# B&R Automation Studio project NAELD004C00R10L518F00 (part 28)

#### Local.var
```iecst
(*2019-06-07*)
(**)
(*Local Action, State & Status*)
VAR
	eAct : eBufferAction := BufferActIdle;
	eStat : eBufferAction := BufferActIdle;
	eStatus : eFBStatus := Idle;
	udiStatus : UDINT := 0;
	sStatTxt : STRING[200] := '';
	a_sStatText : ARRAY[0..50] OF STRING[200] := ['Idling','Creating Directory','Getting Retained Buffer Data','Setting Buffer Full','Setting Buffer Empty','Loading Board','Loading Board With Slot Check','Unloading Board','Unloading Board With Slot Check','Unloading Board With Cooling Time Check','Unloading Board With Slot Check And Cooling Time Check','Getting Next Load Board Slot Number','Getting Next Load Good Board Slot Number','Getting Next Load Bad Board Slot Number','Getting Next Unload Board Slot Number','Getting Next Unload Good Board Slot Number','Getting Next Unload Bad Board Slot Number','Checking Cooling Time','Checking Cooling Board','Checking Cooling Good Board','Checking Cooling Bad Board','Resetting Buffer','Turning On Cooling Fan','Turning Off Cooling Fan','Background Starting Buffer Set Full','Background Starting Buffer Set Empty','Background Stopping Buffer Set','Background Starting Update Sensor','Background Stopping Update Sensor','Background Starting Update Display','Background Stopping Update Display','Background Starting Cooling Fan','Background Stopping Cooling Fan',18('')];
END_VAR
(**)
(*Local Alarm*)
VAR
	tyAlmData : tyAlmDat;
	a_tyAlmText : ARRAY[10000..10099] OF tyAlmTxt := [(sAlmText:='Create User Directory Error',sRcyText:='An Error Occurred While Attempting To Create User Directory. Please Contact Nutek For A Possible Solution'),(sAlmText:='Create Retain Directory Error',sRcyText:='An Error Occurred While Attempting To Create Retain Directory. Please Contact Nutek For A Possible Solution'),(sAlmText:='File Open Error While Reading Retain File',sRcyText:='An Error Was Encountered While Trying To Open File. Please Contact Nutek For A Possible Solution.'),(sAlmText:='File Read Error While Reading Retain File',sRcyText:='An Error Was Encountered While Trying To Read File. Please Contact Nutek For A Possible Solution.'),(sAlmText:='File Close Error While Reading Retain File',sRcyText:='An Error Was Encountered While Trying To Close File. Please Contact Nutek For A Possible Solution.'),(sAlmText:='File Open Error While Setting Full Buffer',sRcyText:='An Error Was Encountered While Trying To Open File. Please Contact Nutek For A Possible Solution.'),(sAlmText:='File Create Error While Setting Full Buffer',sRcyText:='An Error Was Encountered While Trying To Create File. Please Contact Nutek For A Possible Solution.'),(sAlmText:='File Write Error While Setting Full Buffer',sRcyText:='An Error Was Encountered While Trying To Write File. Please Contact Nutek For A Possible Solution.'),(sAlmText:='File Close Error While Setting Full Buffer',sRcyText:='An Error Was Encountered While Trying To Close File. Please Contact Nutek For A Possible Solution.'),(sAlmText:='File Open Error While Setting Empty Buffer',sRcyText:='An Error Was Encountered While Trying To Open File. Please Contact Nutek For A Possible Solution.'),(sAlmText:='File Create Error While Setting Empty Buffer',sRcyText:='An Error Was Encountered While Trying To Create File. Please Contact Nutek For A Possible Solution.'),(sAlmText:='File Write Error While Setting Empty Buffer',sRcyText:='An Error Was Encountered While Trying To Write File. Please Contact Nutek For A Possible Solution.'),(sAlmText:='File Close Error While Setting Empty Buffer',sRcyText:='An Error Was Encountered While Trying To Close File. Please Contact Nutek For A Possible Solution.'),(sAlmText:='File Open Error While Loading Info To Buffer',sRcyText:='An Error Was Encountered While Trying To Open File. Please Contact Nutek For A Possible Solution.'),(sAlmText:='File Create Error While Loading Info To Buffer',sRcyText:='An Error Was Encountered While Trying To Create File. Please Contact Nutek For A Possible Solution.'),(sAlmText:='File Write Error While Loading Info To Buffer',sRcyText:='An Error Was Encountered While Trying To Write File. Please Contact Nutek For A Possible Solution.'),(sAlmText:='File Close Error While Loading Info To Buffer',sRcyText:='An Error Was Encountered While Trying To Close File. Please Contact Nutek For A Possible Solution.'),(sAlmText:='Wrong Slot Number To Load',sRcyText:='Invalid Slot to Load The Board.'),(sAlmText:='File Open Error While Loading Info To Buffer With Slot Check',sRcyText:='An Error Was Encountered While Trying To Open File. Please Contact Nutek For A Possible Solution.'),(sAlmText:='File Create Error While Loading Info To Buffer With Slot Check',sRcyText:='An Error Was Encountered While Trying To Create File. Please Contact Nutek For A Possible Solution.'),(sAlmText:='File Write Error While Loading Info To Buffer With Slot Check',sRcyText:='An Error Was Encountered While Trying To Write File. Please Contact Nutek For A Possible Solution.'),(sAlmText:='File Close Error While Loading Info To Buffer With Slot Check',sRcyText:='An Error Was Encountered While Trying To Close File. Please Contact Nutek For A Possible Solution.'),(sAlmText:='File Open Error While Unloading Info From Buffer',sRcyText:='An Error Was Encountered While Trying To Open File. Please Contact Nutek For A Possible Solution.'),(sAlmText:='File Create Error While Unloading Info From Buffer',sRcyText:='An Error Was Encountered While Trying To Create File. Please Contact Nutek For A Possible Solution.'),(sAlmText:='File Write Error While Unloading Info From Buffer',sRcyText:='An Error Was Encountered While Trying To Write File. Please Contact Nutek For A Possible Solution.'),(sAlmText:='File Close Error While Unloading Info From Buffer',sRcyText:='An Error Was Encountered While Trying To Close File. Please Contact Nutek For A Possible Solution.'),(sAlmText:='Wrong Slot Number To Unload',sRcyText:='Invalid Slot to Unload The Board.'),(sAlmText:='File Open Error While Unloading Info From Buffer With Slot Check',sRcyText:='An Error Was Encountered While Trying To Open File. Please Contact Nutek For A Possible Solution.'),(sAlmText:='File Create Error While Unloading Info From Buffer With Slot Check',sRcyText:='An Error Was Encountered While Trying To Create File. Please Contact Nutek For A Possible Solution.'),(sAlmText:='File Write Error While Unloading Info From Buffer With Slot Check',sRcyText:='An Error Was Encountered While Trying To Write File. Please Contact Nutek For A Possible Solution.'),(sAlmText:='File Close Error While Unloading Info From Buffer With Slot Check',sRcyText:='An Error Was Encountered While Trying To Close File. Please Contact Nutek For A Possible Solution.'),(sAlmText:='File Open Error While Unloading Info From Buffer With Cooling Time Check',sRcyText:='An Error Was Encountered While Trying To Open File. Please Contact Nutek For A Possible Solution.'),(sAlmText:='File Create Error While Unloading Info From Buffer With Cooling Time Check',sRcyText:='An Error Was Encountered While Trying To Create File. Please Contact Nutek For A Possible Solution.'),(sAlmText:='File Write Error While Unloading Info From Buffer With Cooling Time Check',sRcyText:='An Error Was Encountered While Trying To Write File. Please Contact Nutek For A Possible Solution.'),(sAlmText:='File Close Error While Unloading Info From Buffer With Cooling Time Check',sRcyText:='An Error Was Encountered While Trying To Close File. Please Contact Nutek For A Possible Solution.'),(sAlmText:='Wrong Slot Number To Unload With Cooling Time Check',sRcyText:='Invalid Slot to Unload The Board with Cooling Time Check.'),(sAlmText:='File Open Error While Unloading Info From Buffer With Slot Check And Cooling Time Check',sRcyText:='An Error Was Encountered While Trying To Open File. Please Contact Nutek For A Possible Solution.'),(sAlmText:='File Create Error While Unloading Info From Buffer With Slot Check And Cooling Time Check',sRcyText:='An Error Was Encountered While Trying To Create File. Please Contact Nutek For A Possible Solution.'),(sAlmText:='File Write Error While Unloading Info From Buffer With Slot Check And Cooling Time Check',sRcyText:='An Error Was Encountered While Trying To Write File. Please Contact Nutek For A Possible Solution.'),(sAlmText:='File Close Error While Unloading Info From Buffer With Slot Check And Cooling Time Check',sRcyText:='An Error Was Encountered While Trying To Close File. Please Contact Nutek For A Possible Solution.'),(sAlmText:='Directory Does Not Exist While Setting Full Buffer',sRcyText:='The Directory Does Not Exist. Please Contact Nutek For A Possible Solution.'),(sAlmText:='Directory Does Not Exist While Setting Empty Buffer',sRcyText:='The Directory Does Not Exist. Please Contact Nutek For A Possible Solution.'),(sAlmText:='Directory Does Not Exist While Loading Info To Buffer',sRcyText:='The Directory Does Not Exist. Please Contact Nutek For A Possible Solution.'),(sAlmText:='Directory Does Not Exist While Loading Info To Buffer With Slot Check',sRcyText:='The Directory Does Not Exist. Please Contact Nutek For A Possible Solution.'),(sAlmText:='Directory Does Not Exist While Unloading Info From Buffer',sRcyText:='The Directory Does Not Exist. Please Contact Nutek For A Possible Solution.'),(sAlmText:='Directory Does Not Exist While Unloading Info From Buffer With Slot Check',sRcyText:='The Directory Does Not Exist. Please Contact Nutek For A Possible Solution.'),(sAlmText:='Directory Does Not Exist While Unloading Info From Buffer With Cooling Time Check',sRcyText:='The Directory Does Not Exist. Please Contact Nutek For A Possible Solution.'),(sAlmText:='Directory Does Not Exist While Unloading Info From Buffer With Slot Check And Cooling Time Check',sRcyText:='The Directory Does Not Exist. Please Contact Nutek For A Possible Solution.'),(sAlmText:='Unloading Slot Is Skipped While Unloading Buffer',sRcyText:='Unload From Wrong Slot (Skip Slot).'),(sAlmText:='Unloading Slot Is Not For Board While Unloading Buffer',sRcyText:='Unload From Wrong Slot (Not For Board).'),(sAlmText:='Unloading Slot Board Is Not Available While Unloading Buffer',sRcyText:='Unload From Wrong Slot (Board Is Not Available).'),(sAlmText:='Unloading Last Sub Slot Is Not For Board While Unloading Buffer',sRcyText:='Unload From Wrong Slot (Last Sub Slot Is Not For Board).'),(sAlmText:='Unloading Last Sub Slot Has No Board While Unloading Buffer',sRcyText:='Unload From Wrong Slot (Last Sub Slot Has No Board).'),(sAlmText:='Board Quantity In Slot Is 0 While Unloading Buffer',sRcyText:='Unload From Wrong Slot (Board Quantity In Slot = 0).'),(sAlmText:='Board Capacity In Slot Is 0 While Unloading Buffer',sRcyText:='Unload From Wrong Slot (Board Capacity In Slot = 0).'),(sAlmText:='Unloading Slot Is Skipped While Unloading Buffer With Slot Check',sRcyText:='Unload From Wrong Slot (Skip Slot).'),(sAlmText:='Unloading Slot Is Not For Board While Unloading Buffer With Slot Check',sRcyText:='Unload From Wrong Slot (Not For Board).'),(sAlmText:='Unloading Slot Board Is Not available While Unloading Buffer With Slot Check',sRcyText:='Unload From Wrong Slot (Board Is Not Available).'),(sAlmText:='Unloading Last Sub Slot Is Not For Board While Unloading Buffer With Slot Check',sRcyText:='Unload From Wrong Slot (Last Sub Slot Is Not For Board).'),(sAlmText:='Unloading Last Sub Slot Has No Board While Unloading Buffer With Slot Check',sRcyText:='Unload From Wrong Slot (Last Sub Slot Has No Board).'),(sAlmText:='Board Quantity In Slot Is 0 While Unloading Buffer With Slot Check',sRcyText:='Unload From Wrong Slot (Board Quantity In Slot = 0).'),(sAlmText:='Board Capacity In Slot Is 0 While Unloading Buffer With Slot Check',sRcyText:='Unload From Wrong Slot (Board Capacity In Slot = 0).'),(sAlmText:='Unloading Slot Is Skipped While Unloading Buffer With Cool Check',sRcyText:='Unload From Wrong Slot (Skip Slot).'),(sAlmText:='Unloading Slot Is Not For Board While Unloading Buffer With Cool Check',sRcyText:='Unload From Wrong Slot (Not For Board).'),(sAlmText:='Unloading Slot Board Is Not available While Unloading Buffer With Cool Check',sRcyText:='Unload From Wrong Slot (Board Is Not Available).'),(sAlmText:='Unloading Last Sub Slot Is Not For Board While Unloading Buffer With Cool Check',sRcyText:='Unload From Wrong Slot (Last Sub Slot Is Not For Board).'),(sAlmText:='Unloading Last Sub Slot Has No Board While Unloading Buffer With Cool Check',sRcyText:='Unload From Wrong Slot (Last Sub Slot Has No Board).'),(sAlmText:='Board Quantity In Slot Is 0 While Unloading Buffer With Cool Check',sRcyText:='Unload From Wrong Slot (Board Quantity In Slot = 0).'),(sAlmText:='Board Capacity In Slot Is 0 While Unloading Buffer With Cool Check',sRcyText:='Unload From Wrong Slot (Board Capacity In Slot = 0).'),(sAlmText:='Unloading Slot Is Skipped While Unloading Buffer With Cool & Slot Check',sRcyText:='Unload From Wrong Slot (Skip Slot).'),(sAlmText:='Unloading Slot Is Not For Board While Unloading Buffer With Cool & Slot Check',sRcyText:='Unload From Wrong Slot (Not For Board).'),(sAlmText:='Unloading Slot Board Is Not available While Unloading Buffer With Cool & Slot Check',sRcyText:='Unload From Wrong Slot (Board Is Not Available).'),(sAlmText:='Unloading Last Sub Slot Is Not For Board While Unloading Buffer With Cool & Slot Check',sRcyText:='Unload From Wrong Slot (Last Sub Slot Is Not For Board).'),(sAlmText:='Unloading Last Sub Slot Has No Board While Unloading Buffer With Cool & Slot Check',sRcyText:='Unload From Wrong Slot (Last Sub Slot Has No Board).'),(sAlmText:='Board Quantity In Slot Is 0 While Unloading Buffer With Cool & Slot Check',sRcyText:='Unload From Wrong Slot (Board Quantity In Slot = 0).'),(sAlmText:='Board Capacity In Slot Is 0 While Unloading Buffer With Cool & Slot Check',sRcyText:='Unload From Wrong Slot (Board Capacity In Slot = 0).'),(sAlmText:='Loading Slot Is Not For Board',sRcyText:='Load To Wrong Slot (Not For Board).'),(sAlmText:='Loading Slot Is Full Of Board',sRcyText:='Load To Wrong Slot (Full With Board).'),(sAlmText:='Loading First Sub-Slot Is Not For Board',sRcyText:='Load To Wrong Slot (First Sub Slot Not For Board).'),(sAlmText:='Loading Last Sub-Slot Have Board, Which Mean Slot Is Full Of Board',sRcyText:='Load To Wrong Slot (Full With Board(Last Sub Slot Have Board)).'),(sAlmText:='Loading Last Sub-Slot Is Not For Board',sRcyText:='Load To Wrong Slot (Last Sub Slot Not For Board).'),(sAlmText:='Loading Slot Is Full Of Board',sRcyText:='Load To Wrong Slot (Full With Board).'),(sAlmText:='Loading Slot Is Skipped',sRcyText:='Load To Wrong Slot (Skip Slot).'),(sAlmText:='Existing Board Status Is Different With Loading Board Status',sRcyText:='Existing Board Status Is Different With Loading Buffer Status.'),(sAlmText:='Loading Slot Is Not For Board',sRcyText:='Load To Wrong Slot (Not For Board).'),(sAlmText:='Loading Slot Is Full Of Board',sRcyText:='Load To Wrong Slot (Full With Board).'),(sAlmText:='Loading First Sub-Slot Is Not For Board',sRcyText:='Load To Wrong Slot (First Sub Slot Not For Board).'),(sAlmText:='Loading Last Sub-Slot Have Board, Which Mean Slot Is Full Of Board',sRcyText:='Load To Wrong Slot (Full With Board(Last Sub Slot Have Board)).'),(sAlmText:='Loading Last Sub-Slot Is Not For Board',sRcyText:='Load To Wrong Slot (Last Sub Slot Not For Board).'),(sAlmText:='Loading Slot Is Full Of Board',sRcyText:='Load To Wrong Slot (Full With Board).'),(sAlmText:='Loading Slot Is Skipped',sRcyText:='Load To Wrong Slot (Skip Slot).'),(sAlmText:='Existing Board Status Is Different With Loading Board Status',sRcyText:='Existing Board Status Is Different With Loading Buffer Status.'),8((0))];
END_VAR
(**)
(*Local Output*)
VAR
	diNxtLoadSlt : DINT;
	diNxtUnloadSlt : DINT;
	diCoolBrdAny : DINT;
	diCoolBrdGd : DINT;
	diCoolBrdBad : DINT;
	bCoolNotRdy : BOOL;
	tyBuffer : tyBffr;
	tyDispBuffer : tyDispBffr;
	tyBufferStat : tyBffrStat;
	tyBoardUnloadStat : tyBrdUnloadStat;
	bFileNotFound : BOOL;
	bCoolFanCtrl : BOOL;
END_VAR
VAR RETAIN
	bMagPresent : BOOL;
END_VAR
VAR
	dtMagPresentTm : DATE_AND_TIME;
	bNewProduct : BOOL;
	bLastProductUnload : BOOL;
	bLastProductLeftInBffr : BOOL;
	bParamDiff : BOOL;
	bMagRemoved : BOOL;
	bFIFOOld : BOOL;
END_VAR
(**)
(*Local Input*)
VAR
	udiRstErr : UDINT := 0;
	sFileName : STRING[80] := 'Buffer.dat';
	bManual : BOOL := FALSE;
	dtCurrDT : DATE_AND_TIME;
	diMinSlt : DINT;
	diMaxSlt : DINT;
	diPitch : DINT;
	diSltCap : DINT := 1;
	diBffrTtlSlt : DINT;
	diCoolTm : DINT;
	diSltToSltInUM : DINT;
	diLifterBtmPosInUM : DINT;
	diLifterCurrPosInUM : DINT;
	bAscending : BOOL;
	bFIFO : BOOL;
	bGdBrdIn : BOOL;
	bGdBrdReq : BOOL;
	bNxtLoadSeq : BOOL;
	a_bSkip : ARRAY[1..c_diBffrSize] OF BOOL;
	diCoolFanOffDlyTm : DINT := 30000;
	bMagPresentSensor : BOOL;
	bPrepCoolFan : BOOL := TRUE;
	bCoolFanTm : BOOL := TRUE;
	sBffrNm : STRING[15];
	sProdNm : STRING[15];
	sBarcode1 : STRING[80];
	sBarcode2 : STRING[80];
	sCurrRcpNm : {REDUND_UNREPLICABLE} STRING[15];
	sProgNm : STRING[15] := 'Buffer';
	bNtSettingsLoadDone : BOOL := TRUE;
END_VAR
(**)
(*Local*)
VAR
	bRstErr : BOOL;
	udiRstErrOld : UDINT;
	bInitDone : BOOL;
	bInitialDone : BOOL;
	bUpdateSensor : BOOL;
	bBffrSetMty : BOOL;
	bBffrSetFull : BOOL;
	bUpdtDisplay : BOOL;
	usiStep : USINT;
	diCurrSlt : DINT;
	diExpectedSlt : DINT;
	bSetFull : BOOL;
	bSetMty : BOOL;
	bCoolFanRun : BOOL;
	tyBffrParameter : tyBffrParam;
	fbDirCreate1 : fbDirCreate;
	fbDirCreate2 : fbDirCreate;
	fbFileRead1 : fbFileFullRead;
	fbFileWrite1 : fbFileFullWrite;
	fbCoolFanOffDlyTm : TON;
	fbCoolFanOffChkTm : TON := (PT:=T#500ms);
	fbMagAbsentTm : TON := (PT:=T#5s);
	fbMagPresentTm : TON := (PT:=T#8s);
	eStatOld : eBufferAction := BufferActIdle;
	udiModuleNum : UDINT := 2001;
END_VAR
```

#### Act_Alarm.st
```iecst
(** 2019-03-25 **)
ACTION Act_Alarm:

	//Error
	IF EDGEPOS(eStatus = Error) THEN

		tyAlmData.sProgNm		:= p_sProgNm;
		tyAlmData.udiCode		:= udiStatus;
		tyAlmData.eSeverity		:= AlmSeverityError;
		tyAlmData.udiRunTime	:= tyAlmData.udiRunTime + 1;
		tyAlmData.bAlm			:= TRUE;
		tyAlmData.udiModuleNum  := udiModuleNum;
		g_sBufferProgNm		:= p_sProgNm;
		//Get Error Message
		IF tyAlmData.udiCode < 10000 OR tyAlmData.udiCode > 10099 THEN
			tyAlmData.sAlmMsg	:= 'Unknown';
			tyAlmData.sRcyMsg	:= 'Unknown';
		ELSE
			tyAlmData.sAlmMsg	:= a_tyAlmText[tyAlmData.udiCode].sAlmText;
			tyAlmData.sRcyMsg	:= a_tyAlmText[tyAlmData.udiCode].sRcyText;
		END_IF

		sStatTxt	:= tyAlmData.sAlmMsg;

	ELSIF bRstErr AND (tyAlmData.udiCode <> 0) THEN

		tyAlmData.udiCode	:= 0;
		tyAlmData.eSeverity	:= AlmSeverityNA;
		tyAlmData.sAlmMsg	:= '';
		tyAlmData.sRcyMsg	:= '';
		tyAlmData.bAlm			:= FALSE;
		sStatTxt	:= a_sStatText[eStat];

	END_IF

END_ACTION
```

#### Act_Background.st
```iecst
(** 2019-07-03 **)
ACTION Act_Background:

	fbMagPresentTm(IN := p_bMagPresentSensor);

	//Update Retain
	IF bUpdateSensor = TRUE THEN
		bMagPresent	:= fbMagPresentTm.Q;
	END_IF

	//Display Buffer
	IF bUpdtDisplay = TRUE THEN
		fDispBffrDescending(ADR(p_tyDispBuffer) , tyBffrParameter , p_tyBuffer , p_dtCurrDT , DINT_TO_TIME(p_diCoolTm) , 0 , 1 , 2);
	END_IF

	//Cooling Fan Control
	IF p_bManual = TRUE THEN
		;

	ELSIF bCoolFanRun = TRUE AND p_bPrepCoolFan = TRUE AND bCoolFanTm = TRUE THEN //Cooling Fan Control By Cooling Time

		fbCoolFanOffChkTm(IN := TRUE);

		IF fbCoolFanOffChkTm.Q = TRUE THEN
			IF fBffrChkCoolBrdAny(p_dtCurrDT, DINT_TO_TIME(p_diCoolTm), p_tyBuffer) = 0 THEN
				fbCoolFanOffDlyTm.IN	:= TRUE;
			ELSE
				fbCoolFanOffDlyTm.IN	:= FALSE;
				bCoolFanCtrl			:= TRUE;
			END_IF

			fbCoolFanOffChkTm(IN := FALSE);
		END_IF

		fbCoolFanOffDlyTm;

		IF fbCoolFanOffDlyTm.Q = TRUE THEN
			bCoolFanCtrl	:= FALSE;
		END_IF

	ELSIF bCoolFanRun = TRUE AND p_bPrepCoolFan = TRUE AND bCoolFanTm = FALSE THEN	//Cooling Fan Control By Buffer Empty
		fbCoolFanOffDlyTm(IN := p_tyBufferStat.bBffrMty);

		IF p_tyBufferStat.bBffrMty = FALSE THEN
			bCoolFanCtrl	:= TRUE;
		END_IF

		IF fbCoolFanOffDlyTm.Q = TRUE THEN
			bCoolFanCtrl	:= FALSE;
		END_IF

	ELSE

		bCoolFanCtrl	:= FALSE;

	END_IF

	//Set Buffer By Magazine Present
	IF bBffrSetFull = TRUE THEN
		IF p_bMagPresentSensor = TRUE AND fbMagAbsentTm.Q = TRUE THEN
			bSetFull		:= TRUE;
			dtMagPresentTm	:= p_dtCurrDT;
		END_IF

		IF bSetFull = TRUE THEN
			p_eAct	:= BufferActSetFull;

			IF eStatus = Done AND eStat = BufferActSetFull THEN
				p_eAct		:= BufferActIdle;
				bSetFull	:= FALSE;
			ELSIF eStatus = Error THEN
				bSetFull	:= FALSE;
			END_IF
		END_IF

		fbMagAbsentTm(IN := NOT p_bMagPresentSensor);

	ELSIF bBffrSetMty = TRUE THEN
		IF p_bMagPresentSensor = TRUE AND fbMagAbsentTm.Q = TRUE THEN
			bSetMty			:= TRUE;
			dtMagPresentTm	:= p_dtCurrDT;
		END_IF

		IF bSetMty = TRUE THEN
			p_eAct	:= BufferActSetMty;

			IF eStatus = Done AND eStat = BufferActSetMty THEN
				p_eAct	:= BufferActIdle;
				bSetMty	:= FALSE;
			ELSIF eStatus = Error THEN
				bSetMty	:= FALSE;
			END_IF
		END_IF

		fbMagAbsentTm(IN := NOT p_bMagPresentSensor);

	END_IF

	//Check Parameter Different
	bParamDiff	:= (tyBffrParameter.bAscending <> p_bAscending)
	OR (tyBffrParameter.diMinSlt <> p_diMinSlt)
	OR (tyBffrParameter.diMaxSlt <> p_diMaxSlt)
	OR (tyBffrParameter.diPitch <> p_diPitch)
	OR (tyBffrParameter.diSltCap <> p_diSltCap)
	OR (bFIFOOld <> p_bFIFO);

	//Update MagRemoved
	bMagRemoved	:= fbMagAbsentTm.Q;

END_ACTION
```

#### Act_InitGlobal.st
```iecst
(** 2019-04-26 **)
ACTION Act_InitGlobal:

	(* Always Change If Project Change *)

	//Pass Data To Link
	p_bLinkStartupRun ACCESS p_StartupRun;
	p_bLinkNtParamProjMagConvPrep ACCESS p_NtParamProjMag4ConvPrep;
//	p_eLinkOpsMagLDBufferAct ACCESS p_OpsMagLD4BufferAct;
	p_eLinkOpsMagConvLDBufferAct ACCESS p_OpsMagConvLD4BufferAct;

	p_bLinkMcParamProdSelTopToBtm ACCESS p_NtParamProjTopToBtmDefault;//p_ProdRcpCurrRcp1TopToBtm;
	p_bLinkPresentSen1 ACCESS p_DIMagPresentSen4;
	p_bLinkPresentSen2 ACCESS p_DIMagConvEntSen4;

	p_eLinkMag ACCESS p_NtParamProjMag;
	p_usiLinkMod ACCESS p_ProdRcpCurrRcp1McMod;

	p_diLinkSltToSltDist ACCESS p_MagRcpCurrRcpSltToSlt;
	p_diLinkMinSlt ACCESS p_ProdRcpCurrRcp1MinSltValue;
	p_diLinkMaxSlt ACCESS p_ProdRcpCurrRcp1MaxSltValue;
	p_diLinkPitch ACCESS p_ProdRcpCurrRcp1Pitch;
	p_diLinkBffrTtlSlt ACCESS p_MagRcpCurrRcpTtlSlt;
	p_diLinkLifterBtmPosInUM ACCESS p_MagRcpCurrRcpMag4Slt1Pos;

	p_diLinkSltToSltDist1 ACCESS p_MagRcpCurrRcpSltToSlt1;
	p_diLinkMinSlt1 ACCESS p_ProdRcpCurrRcp1MinSltRear;
	p_diLinkMaxSlt1 ACCESS p_ProdRcpCurrRcp1MaxSltRear;
	p_diLinkPitch1 ACCESS p_ProdRcpCurrRcp1PitchRear;
	p_diLinkBffrTtlSlt1 ACCESS p_MagRcpCurrRcpTtlSlt1;
	p_diLinkLifterBtmPosInUM1 ACCESS p_MagRcpCurrRcpMag4Slt1Pos1;

	p_bLinkNtParamProjRotCylPrep ACCESS p_NtParamProjPullerRotCylPrep;

	p_bLinkProjLifterMagPlatform ACCESS p_NtParamProjLifterMagPlatform;
//	p_eLinkOpsLifMagULBufferAct ACCESS p_OpsLifMagLDBufferAct4;
	p_diNtParamProjMagMaxSlt ACCESS p_NtParamProjMagMaxSlt; //initial

	//Pass Data To Internal Use
	p_udiRstErr ACCESS p_RstErrReset;
	p_sFileName ACCESS p_NtParamBffr4FileNm;
	p_bManual ACCESS p_UIMnlMod;
	p_dtCurrDT ACCESS p_TimeCurrDT;
//	p_diMinSlt ACCESS p_ProdRcpCurrRcp1MinSltValue;
//	p_diMaxSlt ACCESS p_ProdRcpCurrRcp1MaxSltValue;
//	p_diPitch ACCESS p_ProdRcpCurrRcp1Pitch;
//	p_diBffrTtlSlt ACCESS p_MagRcpCurrRcpTtlSlt;
//	p_diLifterBtmPosInUM ACCESS p_MagRcpCurrRcpMag4Slt1Pos;
	p_diLifterCurrPosInUM ACCESS p_LifterBtmActualPos;
	p_bFIFO ACCESS p_NtParamBffr4FIFO;
//	p_bMagPresentSensor ACCESS p_DIMagPresentSen4;
	p_sCurrRcpNm ACCESS p_ProdRcpCurrRcp1Nm;
	p_sProgNm ACCESS p_NtParamBffr4ProgNm;
	p_bNtSettingsLoadDone ACCESS p_StartupNtSettingsLoadDone;

	(* Always Change If Project Change *)

END_ACTION
```

#### Act_Link.st
```iecst
(** 2019-03-29 **)
ACTION Act_Link:

	IF p_eLinkMag = LDMagQuadruple THEN
		CASE p_usiLinkMod OF
			0: //LDModLoadLnA:
				IF p_bAscending THEN
					p_diSltToSltInUM := p_diLinkSltToSltDist * -1;
				ELSE
					p_diSltToSltInUM := p_diLinkSltToSltDist;
				END_IF
				p_diMinSlt := p_diLinkMinSlt;
				p_diMaxSlt := p_diLinkMaxSlt;
				p_diPitch := p_diLinkPitch;
				p_diBffrTtlSlt := p_diLinkBffrTtlSlt;
				p_diLifterBtmPosInUM := p_diLinkLifterBtmPosInUM;

			1,2: //LDModLoadLnB, LDModLoadLnAB:
				IF p_bAscending THEN
					p_diSltToSltInUM := p_diLinkSltToSltDist1 * -1;
				ELSE
					p_diSltToSltInUM := p_diLinkSltToSltDist1;
				END_IF
				p_diMinSlt := p_diLinkMinSlt1;
				p_diMaxSlt := p_diLinkMaxSlt1;
				p_diPitch := p_diLinkPitch1;
				p_diBffrTtlSlt := p_diLinkBffrTtlSlt1;
				p_diLifterBtmPosInUM := p_diLinkLifterBtmPosInUM1;

		END_CASE
	ELSE
		IF p_bAscending THEN
			p_diSltToSltInUM := p_diLinkSltToSltDist * -1;
		ELSE
			p_diSltToSltInUM := p_diLinkSltToSltDist;
		END_IF
		p_diMinSlt := p_diLinkMinSlt;
		p_diMaxSlt := p_diLinkMaxSlt;
		p_diPitch := p_diLinkPitch;
		p_diBffrTtlSlt := p_diLinkBffrTtlSlt;
		p_diLifterBtmPosInUM := p_diLinkLifterBtmPosInUM;
	END_IF

	p_bAscending	:= NOT p_bLinkMcParamProdSelTopToBtm;
//	IF p_bLinkNtParamProjRotCylPrep THEN
//		p_bAscending := TRUE;
//	ELSE
//		p_bAscending := FALSE;
//	END_IF

	IF p_bLinkNtParamProjMagConvPrep THEN
		fbMagPresentTm.PT	:= T#2s;
	ELSE
		fbMagPresentTm.PT	:= T#8s;
	END_IF

	p_bMagPresentSensor := p_bLinkPresentSen1 OR p_bLinkPresentSen2;

END_ACTION
```

#### Act_LinkAction.st
```iecst
(** 2019-05-10 **)
ACTION Act_LinkAction:

	IF p_bLinkStartupRun = TRUE THEN
		p_eAct ACCESS p_StartupBuffer4Act;
	ELSE
		IF eStatus = Idle THEN

			IF p_eLinkOpsMagConvLDBufferAct <> BufferActIdle THEN
				p_eAct ACCESS p_OpsMagConvLD4BufferAct;
			ELSE
				p_eAct ACCESS p_UIBuffer4Act;
			END_IF

		END_IF
	END_IF

END_ACTION
```

#### Init.st
```iecst
(** 2019-06-07 **)
PROGRAM _INIT

	(* Always Change If Project Change *)

	//Pass Address To Global Address For External Use
	//Action, State & Status
	p_Buffer4Stat		:= ADR(eStat);
	p_Buffer4Status		:= ADR(eStatus);
	p_Buffer4StatTxt	:= ADR(sStatTxt);

	//Alarm
	p_Buffer4AlmData	:= ADR(tyAlmData);

	//Output
	p_Buffer4NxtLoadSlt				:= ADR(diNxtLoadSlt);
	p_Buffer4NxtUnloadSlt			:= ADR(diNxtUnloadSlt);
	p_Buffer4CoolBrdAny				:= ADR(diCoolBrdAny);
	p_Buffer4CoolBrdGd				:= ADR(diCoolBrdGd);
	p_Buffer4CoolBrdBad				:= ADR(diCoolBrdBad);
	p_Buffer4CoolNotRdy				:= ADR(bCoolNotRdy);
	p_Buffer4Bffr					:= ADR(tyBuffer);
	p_Buffer4DispBffr				:= ADR(tyDispBuffer);
	p_Buffer4BffrStat				:= ADR(tyBufferStat);
	p_Buffer4BrdUnloadStat			:= ADR(tyBoardUnloadStat);
	p_Buffer4FileNotFound			:= ADR(bFileNotFound);
	p_Buffer4CoolFanCtrl			:= ADR(bCoolFanCtrl);
	p_Buffer4MagPresent				:= ADR(bMagPresent);
	p_Buffer4MagPresentTm			:= ADR(dtMagPresentTm);
	p_Buffer4NewProduct				:= ADR(bNewProduct);
	p_Buffer4LastProductUnload		:= ADR(bLastProductUnload);
	p_Buffer4LastProductLeftInBffr	:= ADR(bLastProductLeftInBffr);
	p_Buffer4ParamDiff				:= ADR(bParamDiff);
	p_Buffer4MagRemoved				:= ADR(bMagRemoved);
	p_Buffer4FIFOOld				:= ADR(bFIFOOld);

	(* Always Change If Project Change *)

END_PROGRAM
```

### Program Logical/SMEMA/USSMEMA1 (IEC) - 1.00.0 - NtSMEMA v5.00.0

#### Act_InitGlobal.st
```iecst
(** 2019-04-09 **)
ACTION Act_InitGlobal:

	(* Always Change If Project Change *)

	//Pass Data To Link
	p_bLinkOpsRun ACCESS p_OpsRun;

	p_bLinkNtParamProjPullerRotPrep ACCESS p_NtParamProjPullerRotCylPrep;
	p_bLinkConvHvBrd ACCESS p_PullConvHvBrd;
	p_eLinkConvDir ACCESS p_NtParamProjConvDir;
	p_eLinkOpsTravLifPosGo ACCESS p_OpsTravLifLDPosGo;
	p_bLinkDIPullExtRS ACCESS p_DIPullerExtRS;
	p_bLinkDIPullRetRS ACCESS p_DIPullerRetRS;
	p_diLinkProdRcpCurrRcpPitch ACCESS p_ProdRcpCurrRcp2Pitch;

	//Pass Data To Internal Use
	p_udiRstErr ACCESS p_RstErrReset;
	p_bManual ACCESS p_UIMnlMod;
	p_bLeftSen ACCESS p_DIConvLftSen;
	p_bRightSen ACCESS p_DIConvRgtSen;
	p_bUBA ACCESS p_DSSMEMA1DBA;
	p_bUBAStat ACCESS p_DSSMEMA1DBAStat;
	p_tRstDlyTm ACCESS p_NtParamUSSMEMA1RstDlyTm;
	p_tSigInChkTm ACCESS p_NtParamUSSMEMA1SigInChkTm;
	p_sProgNm ACCESS p_NtParamUSSMEMA1ProgNm;
	p_bNtSettingsLoadDone ACCESS p_StartupNtSettingsLoadDone;

	(* Always Change If Project Change *)

END_ACTION
```

#### Act_Link.st
```iecst
(** 2019-03-29 **)
ACTION Act_Link:

	//Ready Receive
	p_bRdyRcv	:= p_bLinkConvHvBrd = FALSE AND p_eLinkOpsTravLifPosGo = TravLifLDPosUS1;

	//Receive Complete
	IF eStat <> SMEMAActIdle THEN
		IF p_bLinkDIPullExtRS THEN
			bPulled	:= TRUE;
		END_IF

		p_bComplSigOn	:= NOT p_bLeftSen AND bPulled AND p_bLinkDIPullRetRS;
	ELSE
		bPulled			:= FALSE;
		p_bComplSigOn	:= FALSE;
	END_IF

	//Direction
	p_bDirLToR	:= p_eLinkConvDir = ConvDirLToR OR p_eLinkConvDir = ConvDirLToL;

	//Transfer In Timeout (Smaller Than Conveyor Transfer In Timeout)
	IF p_bLinkNtParamProjPullerRotPrep THEN
		diTransferInTO		:= 12000;
	ELSE
		diTransferInTO		:= 20000 + (p_diLinkProdRcpCurrRcpPitch * 125);
	END_IF

END_ACTION
```

#### Act_LinkAction.st
```iecst
(** 2019-04-09 **)
ACTION Act_LinkAction:

	IF p_bLinkOpsRun = TRUE THEN
		p_eAct ACCESS p_OpsTravLifLDUSSMEMAAct1;
	ELSE
		p_eAct ACCESS ADR(eAct);
	END_IF

END_ACTION
```

### Program Logical/SMEMA/USSMEMA2 (IEC) - 1.00.0 - NtSMEMA v5.00.0

#### InputRef_Link.var
```iecst
(*2019-04-09*)
(**)
(*External Data*)
VAR
	p_bLinkOpsRun : REFERENCE TO BOOL;
END_VAR
(**)
VAR
	p_bLinkNtParamProjPullerRotPrep : REFERENCE TO BOOL;
	p_bLinkConvHvBrd : REFERENCE TO BOOL;
	p_eLinkConvDir : REFERENCE TO eConvDir;
	p_eLinkOpsTravLifPosGo : REFERENCE TO eTravLifLDPos;
	p_bLinkDIPullExtRS : REFERENCE TO BOOL;
	p_bLinkDIPullRetRS : REFERENCE TO BOOL;
	p_diLinkProdRcpCurrRcpPitch : REFERENCE TO DINT;
END_VAR
(**)
VAR
	bPulled : BOOL;
END_VAR
```

#### Act_InitGlobal.st
```iecst
(** 2019-04-09 **)
ACTION Act_InitGlobal:

	(* Always Change If Project Change *)

	//Pass Data To Link
	p_bLinkOpsRun ACCESS p_OpsRun;

	p_bLinkNtParamProjPullerRotPrep ACCESS p_NtParamProjPullerRotCylPrep;
	p_bLinkConvHvBrd ACCESS p_PullConvHvBrd;
	p_eLinkConvDir ACCESS p_NtParamProjConvDir;
	p_eLinkOpsTravLifPosGo ACCESS p_OpsTravLifLDPosGo;
	p_bLinkDIPullExtRS ACCESS p_DIPullerExtRS;
	p_bLinkDIPullRetRS ACCESS p_DIPullerRetRS;
	p_diLinkProdRcpCurrRcpPitch ACCESS p_ProdRcpCurrRcp2Pitch;

	//Pass Data To Internal Use
	p_udiRstErr ACCESS p_RstErrReset;
	p_bManual ACCESS p_UIMnlMod;
	p_bLeftSen ACCESS p_DIConvLftSen;
	p_bRightSen ACCESS p_DIConvRgtSen;
	p_bUBA ACCESS p_DSSMEMA2DBA;
	p_bUBAStat ACCESS p_DSSMEMA2DBAStat;
	p_tRstDlyTm ACCESS p_NtParamUSSMEMA2RstDlyTm;
	p_tSigInChkTm ACCESS p_NtParamUSSMEMA2SigInChkTm;
	p_sProgNm ACCESS p_NtParamUSSMEMA2ProgNm;
	p_bNtSettingsLoadDone ACCESS p_StartupNtSettingsLoadDone;

	(* Always Change If Project Change *)

END_ACTION
```

#### Act_Link.st
```iecst
(** 2019-03-29 **)
ACTION Act_Link:

	//Ready Receive
	p_bRdyRcv	:= p_bLinkConvHvBrd = FALSE AND p_eLinkOpsTravLifPosGo = TravLifLDPosUS2;

	//Receive Complete
	IF eStat <> SMEMAActIdle THEN
		IF p_bLinkDIPullExtRS THEN
			bPulled	:= TRUE;
		END_IF

		p_bComplSigOn	:= NOT p_bLeftSen AND bPulled AND p_bLinkDIPullRetRS;
	ELSE
		bPulled			:= FALSE;
		p_bComplSigOn	:= FALSE;
	END_IF

	//Direction
	p_bDirLToR	:= p_eLinkConvDir = ConvDirLToR OR p_eLinkConvDir = ConvDirLToL;

	//Transfer In Timeout (Smaller Than Conveyor Transfer In Timeout)
	IF p_bLinkNtParamProjPullerRotPrep THEN
		diTransferInTO		:= 12000;
	ELSE
		diTransferInTO		:= 20000 + (p_diLinkProdRcpCurrRcpPitch * 125);
	END_IF

END_ACTION
```

#### Act_LinkAction.st
```iecst
(** 2019-04-09 **)
ACTION Act_LinkAction:

	IF p_bLinkOpsRun = TRUE THEN
		p_eAct ACCESS p_OpsTravLifLDUSSMEMAAct2;
	ELSE
		p_eAct ACCESS ADR(eAct);
	END_IF

END_ACTION
```

### Program Logical/SMEMA/USSMEMA3 (IEC) - 1.00.0 - NtSMEMA v5.00.0

#### Act_Alarm.st
```iecst
(** 2019-03-25 **)
ACTION Act_Alarm:

	//Error
	IF EDGEPOS(eStatus = Error) THEN

		tyAlmData.sProgNm		:= p_sProgNm;
		tyAlmData.udiCode		:= udiStatus;
		tyAlmData.eSeverity		:= AlmSeverityError;
		tyAlmData.udiRunTime	:= tyAlmData.udiRunTime + 1;
		tyAlmData.bAlm			:= TRUE;
		tyAlmData.udiModuleNum  := udiModuleNum;
		g_sUSSMEMAProgNm		:= p_sProgNm;
		//Get Error Message
		IF tyAlmData.udiCode < 10000 OR tyAlmData.udiCode > 10099 THEN
			tyAlmData.sAlmMsg	:= 'Unknown';
			tyAlmData.sRcyMsg	:= 'Unknown';
		ELSE
			tyAlmData.sAlmMsg	:= a_tyAlmText[tyAlmData.udiCode].sAlmText;
			tyAlmData.sRcyMsg	:= a_tyAlmText[tyAlmData.udiCode].sRcyText;
		END_IF

		sStatTxt	:= tyAlmData.sAlmMsg;

	ELSIF bRstErr AND (tyAlmData.udiCode <> 0) THEN

		tyAlmData.udiCode	:= 0;
		tyAlmData.eSeverity	:= AlmSeverityNA;
		tyAlmData.sAlmMsg	:= '';
		tyAlmData.sRcyMsg	:= '';
		tyAlmData.bAlm			:= FALSE;
		sStatTxt	:= a_sStatText[eStat];

	END_IF

END_ACTION
```

#### Act_InitGlobal.st
```iecst
(** 2019-04-09 **)
ACTION Act_InitGlobal:

	(* Always Change If Project Change *)

	//Pass Data To Link
	p_bLinkOpsRun ACCESS p_OpsRun;

	p_bLinkNtParamProjPullerRotPrep ACCESS p_NtParamProjPullerRotCylPrep;
	p_bLinkConvHvBrd ACCESS p_PullConvHvBrd;
	p_eLinkConvDir ACCESS p_NtParamProjConvDir;
	p_eLinkOpsTravLifPosGo ACCESS p_OpsTravLifLDPosGo;
	p_bLinkDIPullExtRS ACCESS p_DIPullerExtRS;
	p_bLinkDIPullRetRS ACCESS p_DIPullerRetRS;
	p_diLinkProdRcpCurrRcpPitch ACCESS p_ProdRcpCurrRcp2Pitch;

	//Pass Data To Internal Use
	p_udiRstErr ACCESS p_RstErrReset;
	p_bManual ACCESS p_UIMnlMod;
	p_bLeftSen ACCESS p_DIConvLftSen;
	p_bRightSen ACCESS p_DIConvRgtSen;
	p_bUBA ACCESS p_DSSMEMA3DBA;
	p_bUBAStat ACCESS p_DSSMEMA3DBAStat;
	p_tRstDlyTm ACCESS p_NtParamUSSMEMA3RstDlyTm;
	p_tSigInChkTm ACCESS p_NtParamUSSMEMA3SigInChkTm;
	p_sProgNm ACCESS p_NtParamUSSMEMA3ProgNm;
	p_bNtSettingsLoadDone ACCESS p_StartupNtSettingsLoadDone;

	(* Always Change If Project Change *)

END_ACTION
```

#### Act_Link.st
```iecst
(** 2019-03-29 **)
ACTION Act_Link:

	//Ready Receive
	p_bRdyRcv	:= p_bLinkConvHvBrd = FALSE AND p_eLinkOpsTravLifPosGo = TravLifLDPosUS3;

	//Receive Complete
	IF eStat <> SMEMAActIdle THEN
		IF p_bLinkDIPullExtRS THEN
			bPulled	:= TRUE;
		END_IF

		p_bComplSigOn	:= NOT p_bLeftSen AND bPulled AND p_bLinkDIPullRetRS;
	ELSE
		bPulled			:= FALSE;
		p_bComplSigOn	:= FALSE;
	END_IF

	//Direction
	p_bDirLToR	:= p_eLinkConvDir = ConvDirLToR OR p_eLinkConvDir = ConvDirLToL;

	//Transfer In Timeout (Smaller Than Conveyor Transfer In Timeout)
	IF p_bLinkNtParamProjPullerRotPrep THEN
		diTransferInTO		:= 12000;
	ELSE
		diTransferInTO		:= 20000 + (p_diLinkProdRcpCurrRcpPitch * 125);
	END_IF

END_ACTION
```

#### Act_LinkAction.st
```iecst
(** 2019-04-09 **)
ACTION Act_LinkAction:

	IF p_bLinkOpsRun = TRUE THEN
		p_eAct ACCESS p_OpsTravLifLDUSSMEMAAct3;
	ELSE
		p_eAct ACCESS ADR(eAct);
	END_IF

END_ACTION
```

### USSMEMA4.var - Change By Project
```iecst
(*2019-03-25*)
(**)
(*Action & State & Status*)
VAR
	p_USSMEMA4Stat : UDINT;
	p_USSMEMA4Status : UDINT;
	p_USSMEMA4StatTxt : UDINT;
END_VAR
(**)
(*Alarm*)
VAR
	p_USSMEMA4AlmData : UDINT;
END_VAR
(**)
(*Output*)
VAR
	p_USSMEMA4USRdy : UDINT;
	p_USSMEMA4USGdBrdRdy : UDINT;
	p_USSMEMA4DSRdy : UDINT;
	p_USSMEMA4Transporting : UDINT;
	p_USSMEMA4ConvStart : UDINT;
	p_USSMEMA4ConvStop : UDINT;
	p_USSMEMA4USB : UDINT;
	p_USSMEMA4Timer : UDINT;
	p_USSMEMA4Virtual : UDINT;
END_VAR
```

### Program Logical/SMEMA/USSMEMA4 (IEC) - 1.00.0 - NtSMEMA v5.00.0

#### Act_InitGlobal.st
```iecst
(** 2019-04-09 **)
ACTION Act_InitGlobal:

	(* Always Change If Project Change *)

	//Pass Data To Link
	p_bLinkOpsRun ACCESS p_OpsRun;

	p_bLinkNtParamProjPullerRotPrep ACCESS p_NtParamProjPullerRotCylPrep;
	p_bLinkConvHvBrd ACCESS p_PullConvHvBrd;
	p_eLinkConvDir ACCESS p_NtParamProjConvDir;
	p_eLinkOpsTravLifPosGo ACCESS p_OpsTravLifLDPosGo;
	p_bLinkDIPullExtRS ACCESS p_DIPullerExtRS;
	p_bLinkDIPullRetRS ACCESS p_DIPullerRetRS;
	p_diLinkProdRcpCurrRcpPitch ACCESS p_ProdRcpCurrRcp2Pitch;

	//Pass Data To Internal Use
	p_udiRstErr ACCESS p_RstErrReset;
	p_bManual ACCESS p_UIMnlMod;
	p_bLeftSen ACCESS p_DIConvLftSen;
	p_bRightSen ACCESS p_DIConvRgtSen;
	p_bUBA ACCESS p_DSSMEMA4DBA;
	p_bUBAStat ACCESS p_DSSMEMA4DBAStat;
	p_tRstDlyTm ACCESS p_NtParamUSSMEMA4RstDlyTm;
	p_tSigInChkTm ACCESS p_NtParamUSSMEMA4SigInChkTm;
	p_sProgNm ACCESS p_NtParamUSSMEMA4ProgNm;
	p_bNtSettingsLoadDone ACCESS p_StartupNtSettingsLoadDone;

	(* Always Change If Project Change *)

END_ACTION
```

#### Act_Link.st
```iecst
(** 2019-03-29 **)
ACTION Act_Link:

	//Ready Receive
	p_bRdyRcv	:= p_bLinkConvHvBrd = FALSE AND p_eLinkOpsTravLifPosGo = TravLifLDPosUS4;

	//Receive Complete
	IF eStat <> SMEMAActIdle THEN
		IF p_bLinkDIPullExtRS THEN
			bPulled	:= TRUE;
		END_IF

		p_bComplSigOn	:= NOT p_bLeftSen AND bPulled AND p_bLinkDIPullRetRS;
	ELSE
		bPulled			:= FALSE;
		p_bComplSigOn	:= FALSE;
	END_IF

	//Direction
	p_bDirLToR	:= p_eLinkConvDir = ConvDirLToR OR p_eLinkConvDir = ConvDirLToL;

	//Transfer In Timeout (Smaller Than Conveyor Transfer In Timeout)
	IF p_bLinkNtParamProjPullerRotPrep THEN
		diTransferInTO		:= 12000;
	ELSE
		diTransferInTO		:= 20000 + (p_diLinkProdRcpCurrRcpPitch * 125);
	END_IF

END_ACTION
```

#### Act_LinkAction.st
```iecst
(** 2019-04-09 **)
ACTION Act_LinkAction:

	IF p_bLinkOpsRun = TRUE THEN
		p_eAct ACCESS p_OpsTravLifLDUSSMEMAAct4;
	ELSE
		p_eAct ACCESS ADR(eAct);
	END_IF

END_ACTION
```

#### Init.st
```iecst
(** 2019-03-25 **)
PROGRAM _INIT

	(* Always Change If Project Change *)

	//Physical Configuration
	tyParam.eSelection	:= SMEMASelIPC9851;

	//Pass Address To Global Address For External Use
	//Action, State & Status
	p_USSMEMA4Stat		:= ADR(eStat);
	p_USSMEMA4Status	:= ADR(eStatus);
	p_USSMEMA4StatTxt	:= ADR(sStatTxt);

	//Alarm
	p_USSMEMA4AlmData	:= ADR(tyAlmData);

	//Output
	p_USSMEMA4USRdy			:= ADR(bUSRdy);
	p_USSMEMA4USGdBrdRdy	:= ADR(bUSGdBrdRdy);
	p_USSMEMA4DSRdy			:= ADR(bDSRdy);
	p_USSMEMA4Transporting	:= ADR(bTransporting);
	p_USSMEMA4ConvStart		:= ADR(bConvStart);
	p_USSMEMA4ConvStop		:= ADR(bConvStop);
	p_USSMEMA4USB			:= ADR(bUSB);
	p_USSMEMA4Timer			:= ADR(bTimer);
	p_USSMEMA4Virtual		:= ADR(bVirtual);

	(* Always Change If Project Change *)

END_PROGRAM
```

### DSSMEMA1.var - Change By Project
```iecst
(*2019-03-25*)
(**)
(*Action & State & Status*)
VAR
	p_DSSMEMA1Stat : UDINT;
	p_DSSMEMA1Status : UDINT;
	p_DSSMEMA1StatTxt : UDINT;
END_VAR
(**)
(*Alarm*)
VAR
	p_DSSMEMA1AlmData : UDINT;
END_VAR
(**)
(*Output*)
VAR
	p_DSSMEMA1USRdy : UDINT;
	p_DSSMEMA1USGdBrdRdy : UDINT;
	p_DSSMEMA1DSRdy : UDINT;
	p_DSSMEMA1Transporting : UDINT;
	p_DSSMEMA1ConvStart : UDINT;
	p_DSSMEMA1ConvStop : UDINT;
	p_DSSMEMA1DBA : UDINT;
	p_DSSMEMA1DBAStat : UDINT;
	p_DSSMEMA1Timer : UDINT;
	p_DSSMEMA1Virtual : UDINT;
END_VAR
```

### Program Logical/SMEMA/DSSMEMA1 (IEC) - 1.00.0 - NtSMEMA v5.00.0

#### Act_InitGlobal.st
```iecst
(** 2019-04-09 **)
ACTION Act_InitGlobal:

	(* Always Change If Project Change *)

	//Pass Data To Link
	p_bLinkOpsRun ACCESS p_OpsRun;
	p_bLinkNtParamProjMagConvPrep ACCESS p_NtParamProjMag1ConvPrep;

	p_bLinkNtParamProjPullerRotPrep ACCESS p_NtParamProjPullerRotCylPrep;
	p_eLinkConvDir ACCESS p_NtParamProjConvDir;
//	p_bLinkOpsMagMagBffrAvl ACCESS p_OpsMagLD1MagBffrAvl;
	p_bLinkOpsMagConvMagBffrAvl ACCESS p_OpsMagConvLD1MagBffrAvl;
	p_bLinkDIPullExtRS ACCESS p_DIPullerExtRS;
	p_bLinkDIPullRetRS ACCESS p_DIPullerRetRS;
	p_diLinkProdRcpCurrRcpPitch ACCESS p_ProdRcpCurrRcp2Pitch;

	p_bLinkProjLifterMagPlatform ACCESS p_NtParamProjLifterMagPlatform;
	p_eLinkOpsLifMagLDMagNxtUnload ACCESS p_OpsLifMagLDMagNxtUnload;
	//Pass Data To Internal Use
	p_udiRstErr ACCESS p_RstErrReset;
	p_bManual ACCESS p_UIMnlMod;
	p_bDSB ACCESS p_USSMEMA1USB;
	p_tRstDlyTm ACCESS p_NtParamDSSMEMA1RstDlyTm;
	p_tSigInChkTm ACCESS p_NtParamDSSMEMA1SigInChkTm;
	p_sProgNm ACCESS p_NtParamDSSMEMA1ProgNm;
	p_bNtSettingsLoadDone ACCESS p_StartupNtSettingsLoadDone;

	(* Always Change If Project Change *)

END_ACTION
```

#### Act_Link.st
```iecst
(** 2019-03-29 **)
ACTION Act_Link:

	//Ready Send
	IF p_bLinkProjLifterMagPlatform = FALSE THEN
		p_bRdySend	:= (*p_bLinkOpsMagMagBffrAvl = TRUE OR*) p_bLinkOpsMagConvMagBffrAvl = TRUE;
	ELSE
		p_bRdySend	:= p_eLinkOpsLifMagLDMagNxtUnload = MagNxtUnloadMag1;
	END_IF
	//Send Complete
	IF eStat <> SMEMAActIdle THEN
		IF p_bLinkDIPullExtRS THEN
			bPulled	:= TRUE;
		END_IF

		p_bComplSigOn	:= bPulled AND p_bLinkDIPullRetRS;
	ELSE
		bPulled			:= FALSE;
		p_bComplSigOn	:= FALSE;
	END_IF

	//Direction
	p_bDirLToR	:= p_eLinkConvDir = ConvDirLToR OR p_eLinkConvDir = ConvDirLToL;

	//Transfer Out Timeout (Same As Upstream SMEMA Transfer In Timeout)
	IF p_bLinkNtParamProjPullerRotPrep THEN
		diTransferOutTO		:= 12000;
	ELSE
		diTransferOutTO		:= 20000 + (p_diLinkProdRcpCurrRcpPitch * 125);
	END_IF

END_ACTION
```

#### Act_LinkAction.st
```iecst
(** 2019-04-09 **)
ACTION Act_LinkAction:

	IF p_bLinkOpsRun = TRUE THEN
		IF p_bLinkProjLifterMagPlatform = FALSE THEN
			p_eAct ACCESS p_OpsMagConvLD1DSSMEMAAct;
		ELSE
			p_eAct ACCESS p_OpsLifMagLDDSSMEMAAct1;
		END_IF
	ELSE
		p_eAct ACCESS ADR(eAct);
	END_IF

END_ACTION
```

#### Init.st
```iecst
(** 2019-03-25 **)
PROGRAM _INIT

	(* Always Change If Project Change *)

	//Physical Configuration
	tyParam.eSelection	:= SMEMASelIPC9851;
	bGdBrd				:= TRUE;

	//Pass Address To Global Address For External Use
	//Action, State & Status
	p_DSSMEMA1Stat		:= ADR(eStat);
	p_DSSMEMA1Status	:= ADR(eStatus);
	p_DSSMEMA1StatTxt	:= ADR(sStatTxt);

	//Alarm
	p_DSSMEMA1AlmData	:= ADR(tyAlmData);

	//Output
	p_DSSMEMA1USRdy			:= ADR(bUSRdy);
	p_DSSMEMA1USGdBrdRdy	:= ADR(bUSGdBrdRdy);
	p_DSSMEMA1DSRdy			:= ADR(bDSRdy);
	p_DSSMEMA1Transporting	:= ADR(bTransporting);
	p_DSSMEMA1ConvStart		:= ADR(bConvStart);
	p_DSSMEMA1ConvStop		:= ADR(bConvStop);
	p_DSSMEMA1DBA			:= ADR(bDBA);
	p_DSSMEMA1DBAStat		:= ADR(bDBAStat);
	p_DSSMEMA1Timer			:= ADR(bTimer);
	p_DSSMEMA1Virtual		:= ADR(bVirtual);

	(* Always Change If Project Change *)

END_PROGRAM
```

### DSSMEMA2.var - Change By Project
```iecst
(*2019-03-25*)
(**)
(*Action & State & Status*)
VAR
	p_DSSMEMA2Stat : UDINT;
	p_DSSMEMA2Status : UDINT;
	p_DSSMEMA2StatTxt : UDINT;
END_VAR
(**)
(*Alarm*)
VAR
	p_DSSMEMA2AlmData : UDINT;
END_VAR
(**)
(*Output*)
VAR
	p_DSSMEMA2USRdy : UDINT;
	p_DSSMEMA2USGdBrdRdy : UDINT;
	p_DSSMEMA2DSRdy : UDINT;
	p_DSSMEMA2Transporting : UDINT;
	p_DSSMEMA2ConvStart : UDINT;
	p_DSSMEMA2ConvStop : UDINT;
	p_DSSMEMA2DBA : UDINT;
	p_DSSMEMA2DBAStat : UDINT;
	p_DSSMEMA2Timer : UDINT;
	p_DSSMEMA2Virtual : UDINT;
END_VAR
```

### Program Logical/SMEMA/DSSMEMA2 (IEC) - 1.00.0 - NtSMEMA v5.00.0

#### Act_InitGlobal.st
```iecst
(** 2019-04-09 **)
ACTION Act_InitGlobal:

	(* Always Change If Project Change *)

	//Pass Data To Link
	p_bLinkOpsRun ACCESS p_OpsRun;
	p_bLinkNtParamProjMagConvPrep ACCESS p_NtParamProjMag2ConvPrep;

	p_bLinkNtParamProjPullerRotPrep ACCESS p_NtParamProjPullerRotCylPrep;
	p_eLinkConvDir ACCESS p_NtParamProjConvDir;
//	p_bLinkOpsMagMagBffrAvl ACCESS p_OpsMagLD2MagBffrAvl;
	p_bLinkOpsMagConvMagBffrAvl ACCESS p_OpsMagConvLD2MagBffrAvl;
	p_bLinkDIPullExtRS ACCESS p_DIPullerExtRS;
	p_bLinkDIPullRetRS ACCESS p_DIPullerRetRS;
	p_diLinkProdRcpCurrRcpPitch ACCESS p_ProdRcpCurrRcp2Pitch;

	p_bLinkProjLifterMagPlatform ACCESS p_NtParamProjLifterMagPlatform;
	p_eLinkOpsLifMagLDMagNxtUnload ACCESS p_OpsLifMagLDMagNxtUnload;
	//Pass Data To Internal Use
	p_udiRstErr ACCESS p_RstErrReset;
	p_bManual ACCESS p_UIMnlMod;
	p_bDSB ACCESS p_USSMEMA2USB;
	p_tRstDlyTm ACCESS p_NtParamDSSMEMA2RstDlyTm;
	p_tSigInChkTm ACCESS p_NtParamDSSMEMA2SigInChkTm;
	p_sProgNm ACCESS p_NtParamDSSMEMA2ProgNm;
	p_bNtSettingsLoadDone ACCESS p_StartupNtSettingsLoadDone;

	(* Always Change If Project Change *)

END_ACTION
```

#### Act_Link.st
```iecst
(** 2019-03-29 **)
ACTION Act_Link:

	//Ready Send
	IF p_bLinkProjLifterMagPlatform = FALSE THEN
		p_bRdySend	:= (*p_bLinkOpsMagMagBffrAvl = TRUE OR*) p_bLinkOpsMagConvMagBffrAvl = TRUE;
	ELSE
		p_bRdySend	:= p_eLinkOpsLifMagLDMagNxtUnload = MagNxtUnloadMag2;
	END_IF
	//Send Complete
	IF eStat <> SMEMAActIdle THEN
		IF p_bLinkDIPullExtRS THEN
			bPulled	:= TRUE;
		END_IF

		p_bComplSigOn	:= bPulled AND p_bLinkDIPullRetRS;
	ELSE
		bPulled			:= FALSE;
		p_bComplSigOn	:= FALSE;
	END_IF

	//Direction
	p_bDirLToR	:= p_eLinkConvDir = ConvDirLToR OR p_eLinkConvDir = ConvDirLToL;

	//Transfer Out Timeout (Same As Upstream SMEMA Transfer In Timeout)
	IF p_bLinkNtParamProjPullerRotPrep THEN
		diTransferOutTO		:= 12000;
	ELSE
		diTransferOutTO		:= 20000 + (p_diLinkProdRcpCurrRcpPitch * 125);
	END_IF

END_ACTION
```

#### Act_LinkAction.st
```iecst
(** 2019-04-09 **)
ACTION Act_LinkAction:

	IF p_bLinkOpsRun = TRUE THEN
		IF p_bLinkProjLifterMagPlatform = FALSE THEN
			p_eAct ACCESS p_OpsMagConvLD2DSSMEMAAct;
		ELSE
			p_eAct ACCESS p_OpsLifMagLDDSSMEMAAct2;
		END_IF
	ELSE
		p_eAct ACCESS ADR(eAct);
	END_IF

END_ACTION
```

#### Init.st
```iecst
(** 2019-03-25 **)
PROGRAM _INIT

	(* Always Change If Project Change *)

	//Physical Configuration
	tyParam.eSelection	:= SMEMASelIPC9851;
	bGdBrd				:= TRUE;

	//Pass Address To Global Address For External Use
	//Action, State & Status
	p_DSSMEMA2Stat		:= ADR(eStat);
	p_DSSMEMA2Status	:= ADR(eStatus);
	p_DSSMEMA2StatTxt	:= ADR(sStatTxt);

	//Alarm
	p_DSSMEMA2AlmData	:= ADR(tyAlmData);

	//Output
	p_DSSMEMA2USRdy			:= ADR(bUSRdy);
	p_DSSMEMA2USGdBrdRdy	:= ADR(bUSGdBrdRdy);
	p_DSSMEMA2DSRdy			:= ADR(bDSRdy);
	p_DSSMEMA2Transporting	:= ADR(bTransporting);
	p_DSSMEMA2ConvStart		:= ADR(bConvStart);
	p_DSSMEMA2ConvStop		:= ADR(bConvStop);
	p_DSSMEMA2DBA			:= ADR(bDBA);
	p_DSSMEMA2DBAStat		:= ADR(bDBAStat);
	p_DSSMEMA2Timer			:= ADR(bTimer);
	p_DSSMEMA2Virtual		:= ADR(bVirtual);

	(* Always Change If Project Change *)

END_PROGRAM
```

### DSSMEMA3.var - Change By Project
```iecst
(*2019-03-25*)
(**)
(*Action & State & Status*)
VAR
	p_DSSMEMA3Stat : UDINT;
	p_DSSMEMA3Status : UDINT;
	p_DSSMEMA3StatTxt : UDINT;
END_VAR
(**)
(*Alarm*)
VAR
	p_DSSMEMA3AlmData : UDINT;
END_VAR
(**)
(*Output*)
VAR
	p_DSSMEMA3USRdy : UDINT;
	p_DSSMEMA3USGdBrdRdy : UDINT;
	p_DSSMEMA3DSRdy : UDINT;
	p_DSSMEMA3Transporting : UDINT;
	p_DSSMEMA3ConvStart : UDINT;
	p_DSSMEMA3ConvStop : UDINT;
	p_DSSMEMA3DBA : UDINT;
	p_DSSMEMA3DBAStat : UDINT;
	p_DSSMEMA3Timer : UDINT;
	p_DSSMEMA3Virtual : UDINT;
END_VAR
```

### Program Logical/SMEMA/DSSMEMA3 (IEC) - 1.00.0 - NtSMEMA v5.00.0

#### InputRef_Link.var
```iecst
(*2019-04-09*)
(**)
(*External Data*)
VAR
	p_bLinkOpsRun : REFERENCE TO BOOL;
	p_bLinkNtParamProjMagConvPrep : REFERENCE TO BOOL;
END_VAR
(**)
VAR
	p_bLinkNtParamProjPullerRotPrep : REFERENCE TO BOOL;
	p_eLinkConvDir : REFERENCE TO eConvDir;
	p_bLinkOpsMagMagBffrAvl : REFERENCE TO BOOL;
	p_bLinkOpsMagConvMagBffrAvl : REFERENCE TO BOOL;
	p_bLinkDIPullExtRS : REFERENCE TO BOOL;
	p_bLinkDIPullRetRS : REFERENCE TO BOOL;
	p_diLinkProdRcpCurrRcpPitch : REFERENCE TO DINT;
	p_bLinkProjLifterMagPlatform : REFERENCE TO BOOL;
	p_eLinkOpsLifMagLDMagNxtUnload : REFERENCE TO eLifMagLDMagNxtUnload;
END_VAR
(**)
VAR
	bPulled : BOOL;
END_VAR
```

#### Act_Alarm.st
```iecst
(** 2019-03-25 **)
ACTION Act_Alarm:

	//Error
	IF EDGEPOS(eStatus = Error) THEN

		tyAlmData.sProgNm		:= p_sProgNm;
		tyAlmData.udiCode		:= udiStatus;
		tyAlmData.eSeverity		:= AlmSeverityError;
		tyAlmData.udiRunTime	:= tyAlmData.udiRunTime + 1;
		tyAlmData.bAlm			:= TRUE;
		tyAlmData.udiModuleNum  := udiModuleNum;
		g_sDSSMEMAProgNm		:= p_sProgNm;
		//Get Error Message
		IF tyAlmData.udiCode < 10000 OR tyAlmData.udiCode > 10099 THEN
			tyAlmData.sAlmMsg	:= 'Unknown';
			tyAlmData.sRcyMsg	:= 'Unknown';
		ELSE
			tyAlmData.sAlmMsg	:= a_tyAlmText[tyAlmData.udiCode].sAlmText;
			tyAlmData.sRcyMsg	:= a_tyAlmText[tyAlmData.udiCode].sRcyText;
		END_IF

		sStatTxt	:= tyAlmData.sAlmMsg;

	ELSIF bRstErr AND (tyAlmData.udiCode <> 0) THEN

		tyAlmData.udiCode	:= 0;
		tyAlmData.eSeverity	:= AlmSeverityNA;
		tyAlmData.sAlmMsg	:= '';
		tyAlmData.sRcyMsg	:= '';
		tyAlmData.bAlm			:= FALSE;
		sStatTxt	:= a_sStatText[eStat];

	END_IF

END_ACTION
```

#### Act_InitGlobal.st
```iecst
(** 2019-04-09 **)
ACTION Act_InitGlobal:

	(* Always Change If Project Change *)

	//Pass Data To Link
	p_bLinkOpsRun ACCESS p_OpsRun;
	p_bLinkNtParamProjMagConvPrep ACCESS p_NtParamProjMag3ConvPrep;

	p_bLinkNtParamProjPullerRotPrep ACCESS p_NtParamProjPullerRotCylPrep;
	p_eLinkConvDir ACCESS p_NtParamProjConvDir;
//	p_bLinkOpsMagMagBffrAvl ACCESS p_OpsMagLD3MagBffrAvl;
	p_bLinkOpsMagConvMagBffrAvl ACCESS p_OpsMagConvLD3MagBffrAvl;
	p_bLinkDIPullExtRS ACCESS p_DIPullerExtRS;
	p_bLinkDIPullRetRS ACCESS p_DIPullerRetRS;
	p_diLinkProdRcpCurrRcpPitch ACCESS p_ProdRcpCurrRcp2Pitch;

	p_bLinkProjLifterMagPlatform ACCESS p_NtParamProjLifterMagPlatform;
	p_eLinkOpsLifMagLDMagNxtUnload ACCESS p_OpsLifMagLDMagNxtUnload;
	//Pass Data To Internal Use
	p_udiRstErr ACCESS p_RstErrReset;
	p_bManual ACCESS p_UIMnlMod;
	p_bDSB ACCESS p_USSMEMA3USB;
	p_tRstDlyTm ACCESS p_NtParamDSSMEMA3RstDlyTm;
	p_tSigInChkTm ACCESS p_NtParamDSSMEMA3SigInChkTm;
	p_sProgNm ACCESS p_NtParamDSSMEMA3ProgNm;
	p_bNtSettingsLoadDone ACCESS p_StartupNtSettingsLoadDone;

	(* Always Change If Project Change *)

END_ACTION
```

#### Act_Link.st
```iecst
(** 2019-03-29 **)
ACTION Act_Link:

	//Ready Send
	IF p_bLinkProjLifterMagPlatform = FALSE THEN
		p_bRdySend	:= (*p_bLinkOpsMagMagBffrAvl = TRUE OR*) p_bLinkOpsMagConvMagBffrAvl = TRUE;
	ELSE
		p_bRdySend	:= p_eLinkOpsLifMagLDMagNxtUnload = MagNxtUnloadMag3;
	END_IF

	//Send Complete
	IF eStat <> SMEMAActIdle THEN
		IF p_bLinkDIPullExtRS THEN
			bPulled	:= TRUE;
		END_IF

		p_bComplSigOn	:= bPulled AND p_bLinkDIPullRetRS;
	ELSE
		bPulled			:= FALSE;
		p_bComplSigOn	:= FALSE;
	END_IF

	//Direction
	p_bDirLToR	:= p_eLinkConvDir = ConvDirLToR OR p_eLinkConvDir = ConvDirLToL;

	//Transfer Out Timeout (Same As Upstream SMEMA Transfer In Timeout)
	IF p_bLinkNtParamProjPullerRotPrep THEN
		diTransferOutTO		:= 12000;
	ELSE
		diTransferOutTO		:= 20000 + (p_diLinkProdRcpCurrRcpPitch * 125);
	END_IF

END_ACTION
```

#### Act_LinkAction.st
```iecst
(** 2019-04-09 **)
ACTION Act_LinkAction:

	IF p_bLinkOpsRun = TRUE THEN
		IF p_bLinkProjLifterMagPlatform = FALSE THEN
			p_eAct ACCESS p_OpsMagConvLD3DSSMEMAAct;
		ELSE
			p_eAct ACCESS p_OpsLifMagLDDSSMEMAAct3;
		END_IF
	ELSE
		p_eAct ACCESS ADR(eAct);
	END_IF

END_ACTION
```

#### Init.st
```iecst
(** 2019-03-25 **)
PROGRAM _INIT

	(* Always Change If Project Change *)

	//Physical Configuration
	tyParam.eSelection	:= SMEMASelIPC9851;
	bGdBrd				:= TRUE;

	//Pass Address To Global Address For External Use
	//Action, State & Status
	p_DSSMEMA3Stat		:= ADR(eStat);
	p_DSSMEMA3Status	:= ADR(eStatus);
	p_DSSMEMA3StatTxt	:= ADR(sStatTxt);

	//Alarm
	p_DSSMEMA3AlmData	:= ADR(tyAlmData);

	//Output
	p_DSSMEMA3USRdy			:= ADR(bUSRdy);
	p_DSSMEMA3USGdBrdRdy	:= ADR(bUSGdBrdRdy);
	p_DSSMEMA3DSRdy			:= ADR(bDSRdy);
	p_DSSMEMA3Transporting	:= ADR(bTransporting);
	p_DSSMEMA3ConvStart		:= ADR(bConvStart);
	p_DSSMEMA3ConvStop		:= ADR(bConvStop);
	p_DSSMEMA3DBA			:= ADR(bDBA);
	p_DSSMEMA3DBAStat		:= ADR(bDBAStat);
	p_DSSMEMA3Timer			:= ADR(bTimer);
	p_DSSMEMA3Virtual		:= ADR(bVirtual);

	(* Always Change If Project Change *)

END_PROGRAM
```

### DSSMEMA4.var - Change By Project
```iecst
(*2019-03-25*)
(**)
(*Action & State & Status*)
VAR
	p_DSSMEMA4Stat : UDINT;
	p_DSSMEMA4Status : UDINT;
	p_DSSMEMA4StatTxt : UDINT;
END_VAR
(**)
(*Alarm*)
VAR
	p_DSSMEMA4AlmData : UDINT;
END_VAR
(**)
(*Output*)
VAR
	p_DSSMEMA4USRdy : UDINT;
	p_DSSMEMA4USGdBrdRdy : UDINT;
	p_DSSMEMA4DSRdy : UDINT;
	p_DSSMEMA4Transporting : UDINT;
	p_DSSMEMA4ConvStart : UDINT;
	p_DSSMEMA4ConvStop : UDINT;
	p_DSSMEMA4DBA : UDINT;
	p_DSSMEMA4DBAStat : UDINT;
	p_DSSMEMA4Timer : UDINT;
	p_DSSMEMA4Virtual : UDINT;
END_VAR
```

### Program Logical/SMEMA/DSSMEMA4 (IEC) - 1.00.0 - NtSMEMA v5.00.0

#### Act_Alarm.st
```iecst
(** 2019-03-25 **)
ACTION Act_Alarm:

	//Error
	IF EDGEPOS(eStatus = Error) THEN

		tyAlmData.sProgNm		:= p_sProgNm;
		tyAlmData.udiCode		:= udiStatus;
		tyAlmData.eSeverity		:= AlmSeverityError;
		tyAlmData.udiRunTime	:= tyAlmData.udiRunTime + 1;
		tyAlmData.bAlm			:= TRUE;
		tyAlmData.udiModuleNum  := udiModuleNum;
		g_sDSSMEMAProgNm		:= p_sProgNm;
		//Get Error Message
		IF tyAlmData.udiCode < 10000 OR tyAlmData.udiCode > 10099 THEN
			tyAlmData.sAlmMsg	:= 'Unknown';
			tyAlmData.sRcyMsg	:= 'Unknown';
		ELSE
			tyAlmData.sAlmMsg	:= a_tyAlmText[tyAlmData.udiCode].sAlmText;
			tyAlmData.sRcyMsg	:= a_tyAlmText[tyAlmData.udiCode].sRcyText;
		END_IF

		sStatTxt	:= tyAlmData.sAlmMsg;

	ELSIF bRstErr AND (tyAlmData.udiCode <> 0) THEN

		tyAlmData.udiCode	:= 0;
		tyAlmData.eSeverity	:= AlmSeverityNA;
		tyAlmData.sAlmMsg	:= '';
		tyAlmData.sRcyMsg	:= '';
		tyAlmData.bAlm			:= FALSE;
		sStatTxt	:= a_sStatText[eStat];

	END_IF

END_ACTION
```

#### Act_InitGlobal.st
```iecst
(** 2019-04-09 **)
ACTION Act_InitGlobal:

	(* Always Change If Project Change *)

	//Pass Data To Link
	p_bLinkOpsRun ACCESS p_OpsRun;
	p_bLinkNtParamProjMagConvPrep ACCESS p_NtParamProjMag4ConvPrep;

	p_bLinkNtParamProjPullerRotPrep ACCESS p_NtParamProjPullerRotCylPrep;
	p_eLinkConvDir ACCESS p_NtParamProjConvDir;
//	p_bLinkOpsMagMagBffrAvl ACCESS p_OpsMagLD4MagBffrAvl;
	p_bLinkOpsMagConvMagBffrAvl ACCESS p_OpsMagConvLD4MagBffrAvl;
	p_bLinkDIPullExtRS ACCESS p_DIPullerExtRS;
	p_bLinkDIPullRetRS ACCESS p_DIPullerRetRS;
	p_diLinkProdRcpCurrRcpPitch ACCESS p_ProdRcpCurrRcp2Pitch;

	p_bLinkProjLifterMagPlatform ACCESS p_NtParamProjLifterMagPlatform;
	p_eLinkOpsLifMagLDMagNxtUnload ACCESS p_OpsLifMagLDMagNxtUnload;
	//Pass Data To Internal Use
	p_udiRstErr ACCESS p_RstErrReset;
	p_bManual ACCESS p_UIMnlMod;
	p_bDSB ACCESS p_USSMEMA4USB;
	p_tRstDlyTm ACCESS p_NtParamDSSMEMA4RstDlyTm;
	p_tSigInChkTm ACCESS p_NtParamDSSMEMA4SigInChkTm;
	p_sProgNm ACCESS p_NtParamDSSMEMA4ProgNm;
	p_bNtSettingsLoadDone ACCESS p_StartupNtSettingsLoadDone;

	(* Always Change If Project Change *)

END_ACTION
```

#### Act_Link.st
```iecst
(** 2019-03-29 **)
ACTION Act_Link:

	//Ready Send
	IF p_bLinkProjLifterMagPlatform = FALSE THEN
		p_bRdySend	:= (*p_bLinkOpsMagMagBffrAvl = TRUE OR*) p_bLinkOpsMagConvMagBffrAvl = TRUE;
	ELSE
//		p_bRdySend	:= p_eLinkOpsLifMagLDMagNxtUnload = MagNxtUnloadMag4;
	END_IF

	//Send Complete
	IF eStat <> SMEMAActIdle THEN
		IF p_bLinkDIPullExtRS THEN
			bPulled	:= TRUE;
		END_IF

		p_bComplSigOn	:= bPulled AND p_bLinkDIPullRetRS;
	ELSE
		bPulled			:= FALSE;
		p_bComplSigOn	:= FALSE;
	END_IF

	//Direction
	p_bDirLToR	:= p_eLinkConvDir = ConvDirLToR OR p_eLinkConvDir = ConvDirLToL;

	//Transfer Out Timeout (Same As Upstream SMEMA Transfer In Timeout)
	IF p_bLinkNtParamProjPullerRotPrep THEN
		diTransferOutTO		:= 12000;
	ELSE
		diTransferOutTO		:= 20000 + (p_diLinkProdRcpCurrRcpPitch * 125);
	END_IF

END_ACTION
```

#### Act_LinkAction.st
```iecst
(** 2019-04-09 **)
ACTION Act_LinkAction:

	IF p_bLinkOpsRun = TRUE THEN
//		IF p_bLinkNtParamProjMagConvPrep = TRUE THEN
			p_eAct ACCESS p_OpsMagConvLD4DSSMEMAAct;
//		ELSE
//			p_eAct ACCESS p_OpsMagLD4DSSMEMAAct;
//		END_IF
	ELSE
		p_eAct ACCESS ADR(eAct);
	END_IF

END_ACTION
```

#### Init.st
```iecst
(** 2019-03-25 **)
PROGRAM _INIT

	(* Always Change If Project Change *)

	//Physical Configuration
	tyParam.eSelection	:= SMEMASelIPC9851;
	bGdBrd				:= TRUE;

	//Pass Address To Global Address For External Use
	//Action, State & Status
	p_DSSMEMA4Stat		:= ADR(eStat);
	p_DSSMEMA4Status	:= ADR(eStatus);
	p_DSSMEMA4StatTxt	:= ADR(sStatTxt);

	//Alarm
	p_DSSMEMA4AlmData	:= ADR(tyAlmData);

	//Output
	p_DSSMEMA4USRdy			:= ADR(bUSRdy);
	p_DSSMEMA4USGdBrdRdy	:= ADR(bUSGdBrdRdy);
	p_DSSMEMA4DSRdy			:= ADR(bDSRdy);
	p_DSSMEMA4Transporting	:= ADR(bTransporting);
	p_DSSMEMA4ConvStart		:= ADR(bConvStart);
	p_DSSMEMA4ConvStop		:= ADR(bConvStop);
	p_DSSMEMA4DBA			:= ADR(bDBA);
	p_DSSMEMA4DBAStat		:= ADR(bDBAStat);
	p_DSSMEMA4Timer			:= ADR(bTimer);
	p_DSSMEMA4Virtual		:= ADR(bVirtual);

	(* Always Change If Project Change *)

END_PROGRAM
```

### DSSMEMAA.var - Change By Project
```iecst
(*2019-03-25*)
(**)
(*Action & State & Status*)
VAR
	p_DSSMEMAAStat : UDINT;
	p_DSSMEMAAStatus : UDINT;
	p_DSSMEMAAStatTxt : UDINT;
END_VAR
(**)
(*Alarm*)
VAR
	p_DSSMEMAAAlmData : UDINT;
END_VAR
(**)
(*Output*)
VAR
	p_DSSMEMAAUSRdy : UDINT;
	p_DSSMEMAAUSGdBrdRdy : UDINT;
	p_DSSMEMAADSRdy : UDINT;
	p_DSSMEMAATransporting : UDINT;
	p_DSSMEMAAConvStart : UDINT;
	p_DSSMEMAAConvStop : UDINT;
	p_DSSMEMAADBA : UDINT;
	p_DSSMEMAADBAStat : UDINT;
	p_DSSMEMAATimer : UDINT;
	p_DSSMEMAAVirtual : UDINT;
END_VAR
```

### Program Logical/SMEMA/DSSMEMAA (IEC) - 1.00.0 - NtSMEMA v5.00.0

#### Act_InitGlobal.st
```iecst
(** 2019-04-09 **)
ACTION Act_InitGlobal:

	(* Always Change If Project Change *)

	//Pass Data To Link
	p_bLinkOpsRun ACCESS p_OpsRun;

	p_bLinkConvHvBrd ACCESS p_PullConvHvBrd;
	p_eLinkConvDir ACCESS p_NtParamProjConvDir;
	p_eLinkOpsTravLifPosGo ACCESS p_OpsTravLifLDPosGo;
	p_bLinkNtParamDSWidthChkPrep ACCESS p_NtParamDSWidthChkPrep;
	p_bLinkMcParamDSWidthChkEn ACCESS p_McParamDSWidthChkEn;
	p_bLinkDIDSWidthChkSen ACCESS p_DIDSWidthChkSen;

	//Pass Data To Internal Use
	p_udiRstErr ACCESS p_RstErrReset;
	p_bManual ACCESS p_UIMnlMod;
	p_tyParam ACCESS p_McParamDSSMEMAAParam;
	p_bGdBrd ACCESS p_PullConvGdBrd;
	p_diTransferOutTO ACCESS p_McParamTranOutErrDlyTm;
	p_bLeftSen ACCESS p_DIConvLftSen;
	p_bRightSen ACCESS p_DIConvRgtSen;
	p_bDSB ACCESS p_DIDSBA;
	p_bVirtualEn ACCESS p_UIVSMEMADSEnA;
	p_bDSBVirtual ACCESS p_UIVSMEMADSBA;
	p_tRstDlyTm ACCESS p_NtParamDSSMEMAARstDlyTm;
	p_tSigInChkTm ACCESS p_NtParamDSSMEMAASigInChkTm;
	p_sProgNm ACCESS p_NtParamDSSMEMAAProgNm;
	p_bNtSettingsLoadDone ACCESS p_StartupNtSettingsLoadDone;

	(* Always Change If Project Change *)

END_ACTION
```

#### Act_Link.st
```iecst
(** 2019-03-29 **)
ACTION Act_Link:

	//Ready Send
	IF p_bLinkNtParamDSWidthChkPrep AND p_bLinkMcParamDSWidthChkEn THEN
		p_bRdySend	:= p_bLinkDIDSWidthChkSen AND p_bLinkConvHvBrd = TRUE AND p_eLinkOpsTravLifPosGo = TravLifLDPosDS1;
	ELSE
		p_bRdySend	:= p_bLinkConvHvBrd = TRUE AND p_eLinkOpsTravLifPosGo = TravLifLDPosDS1;
	END_IF

	//Send Complete
	p_bComplSigOn	:= p_bLinkConvHvBrd = FALSE;

	//Direction
	p_bDirLToR	:= p_eLinkConvDir = ConvDirLToR OR p_eLinkConvDir = ConvDirLToL;

END_ACTION
```

#### Act_LinkAction.st
```iecst
(** 2019-04-09 **)
ACTION Act_LinkAction:

	IF p_bLinkOpsRun = TRUE THEN
		p_eAct ACCESS p_OpsTravLifLDDSSMEMAAct1;
	ELSIF p_bManual = TRUE THEN
		p_eAct ACCESS p_UIDSSMEMAAAct;
	ELSE
		p_eAct ACCESS ADR(eAct);
	END_IF

END_ACTION
```

#### Init.st
```iecst
(** 2019-03-25 **)
PROGRAM _INIT

	(* Always Change If Project Change *)

	//Pass Address To Global Address For External Use
	//Action, State & Status
	p_DSSMEMAAStat		:= ADR(eStat);
	p_DSSMEMAAStatus	:= ADR(eStatus);
	p_DSSMEMAAStatTxt	:= ADR(sStatTxt);

	//Alarm
	p_DSSMEMAAAlmData	:= ADR(tyAlmData);

	//Output
	p_DSSMEMAAUSRdy			:= ADR(bUSRdy);
	p_DSSMEMAAUSGdBrdRdy	:= ADR(bUSGdBrdRdy);
	p_DSSMEMAADSRdy			:= ADR(bDSRdy);
	p_DSSMEMAATransporting	:= ADR(bTransporting);
	p_DSSMEMAAConvStart		:= ADR(bConvStart);
	p_DSSMEMAAConvStop		:= ADR(bConvStop);
	p_DSSMEMAADBA			:= ADR(bDBA);
	p_DSSMEMAADBAStat		:= ADR(bDBAStat);
	p_DSSMEMAATimer			:= ADR(bTimer);
	p_DSSMEMAAVirtual		:= ADR(bVirtual);

	(* Always Change If Project Change *)

END_PROGRAM
```

### DSSMEMAB.var - Change By Project
```iecst
(*2019-03-25*)
(**)
(*Action & State & Status*)
VAR
	p_DSSMEMABStat : UDINT;
	p_DSSMEMABStatus : UDINT;
	p_DSSMEMABStatTxt : UDINT;
END_VAR
(**)
(*Alarm*)
VAR
	p_DSSMEMABAlmData : UDINT;
END_VAR
(**)
(*Output*)
VAR
	p_DSSMEMABUSRdy : UDINT;
	p_DSSMEMABUSGdBrdRdy : UDINT;
	p_DSSMEMABDSRdy : UDINT;
	p_DSSMEMABTransporting : UDINT;
	p_DSSMEMABConvStart : UDINT;
	p_DSSMEMABConvStop : UDINT;
	p_DSSMEMABDBA : UDINT;
	p_DSSMEMABDBAStat : UDINT;
	p_DSSMEMABTimer : UDINT;
	p_DSSMEMABVirtual : UDINT;
END_VAR
```

### Program Logical/SMEMA/DSSMEMAB (IEC) - 1.00.0 - NtSMEMA v5.00.0

#### InputRef_Link.var
```iecst
(*2019-04-09*)
(**)
(*External Data*)
VAR
	p_bLinkOpsRun : REFERENCE TO BOOL;
END_VAR
(**)
VAR
	p_bLinkConvHvBrd : REFERENCE TO BOOL;
	p_eLinkConvDir : REFERENCE TO eConvDir;
	p_eLinkOpsTravLifPosGo : REFERENCE TO eTravLifLDPos;
	p_bLinkNtParamDSWidthChkPrep : REFERENCE TO BOOL;
	p_bLinkMcParamDSWidthChkEn : REFERENCE TO BOOL;
	p_bLinkDIDSWidthChkSen : REFERENCE TO BOOL;
END_VAR
```

#### Act_InitGlobal.st
```iecst
(** 2019-04-09 **)
ACTION Act_InitGlobal:

	(* Always Change If Project Change *)

	//Pass Data To Link
	p_bLinkOpsRun ACCESS p_OpsRun;

	p_bLinkConvHvBrd ACCESS p_PullConvHvBrd;
	p_eLinkConvDir ACCESS p_NtParamProjConvDir;
	p_eLinkOpsTravLifPosGo ACCESS p_OpsTravLifLDPosGo;
	p_bLinkNtParamDSWidthChkPrep ACCESS p_NtParamDSWidthChkPrep;
	p_bLinkMcParamDSWidthChkEn ACCESS p_McParamDSWidthChkEn;
	p_bLinkDIDSWidthChkSen ACCESS p_DIDSWidthChkSen;

	//Pass Data To Internal Use
	p_udiRstErr ACCESS p_RstErrReset;
	p_bManual ACCESS p_UIMnlMod;
	p_tyParam ACCESS p_McParamDSSMEMABParam;
	p_bGdBrd ACCESS p_PullConvGdBrd;
	p_diTransferOutTO ACCESS p_McParamTranOutErrDlyTm;
	p_bLeftSen ACCESS p_DIConvLftSen;
	p_bRightSen ACCESS p_DIConvRgtSen;
	p_bDSB ACCESS p_DIDSBB;
	p_bVirtualEn ACCESS p_UIVSMEMADSEnB;
	p_bDSBVirtual ACCESS p_UIVSMEMADSBB;
	p_tRstDlyTm ACCESS p_NtParamDSSMEMABRstDlyTm;
	p_tSigInChkTm ACCESS p_NtParamDSSMEMABSigInChkTm;
	p_sProgNm ACCESS p_NtParamDSSMEMABProgNm;
	p_bNtSettingsLoadDone ACCESS p_StartupNtSettingsLoadDone;

	(* Always Change If Project Change *)

END_ACTION
```

#### Act_Link.st
```iecst
(** 2019-03-29 **)
ACTION Act_Link:

	//Ready Send
	IF p_bLinkNtParamDSWidthChkPrep AND p_bLinkMcParamDSWidthChkEn THEN
		p_bRdySend	:= p_bLinkDIDSWidthChkSen AND p_bLinkConvHvBrd = TRUE AND p_eLinkOpsTravLifPosGo = TravLifLDPosDS2;
	ELSE
		p_bRdySend	:= p_bLinkConvHvBrd = TRUE AND p_eLinkOpsTravLifPosGo = TravLifLDPosDS2;
	END_IF

	//Send Complete
	p_bComplSigOn	:= p_bLinkConvHvBrd = FALSE;

	//Direction
	p_bDirLToR	:= p_eLinkConvDir = ConvDirLToR OR p_eLinkConvDir = ConvDirLToL;

END_ACTION
```

#### Act_LinkAction.st
```iecst
(** 2019-04-09 **)
ACTION Act_LinkAction:

	IF p_bLinkOpsRun = TRUE THEN
		p_eAct ACCESS p_OpsTravLifLDDSSMEMAAct2;
	ELSIF p_bManual = TRUE THEN
		p_eAct ACCESS p_UIDSSMEMABAct;
	ELSE
		p_eAct ACCESS ADR(eAct);
	END_IF

END_ACTION
```

#### Init.st
```iecst
(** 2019-03-25 **)
PROGRAM _INIT

	(* Always Change If Project Change *)

	//Pass Address To Global Address For External Use
	//Action, State & Status
	p_DSSMEMABStat		:= ADR(eStat);
	p_DSSMEMABStatus	:= ADR(eStatus);
	p_DSSMEMABStatTxt	:= ADR(sStatTxt);

	//Alarm
	p_DSSMEMABAlmData	:= ADR(tyAlmData);

	//Output
	p_DSSMEMABUSRdy			:= ADR(bUSRdy);
	p_DSSMEMABUSGdBrdRdy	:= ADR(bUSGdBrdRdy);
	p_DSSMEMABDSRdy			:= ADR(bDSRdy);
	p_DSSMEMABTransporting	:= ADR(bTransporting);
	p_DSSMEMABConvStart		:= ADR(bConvStart);
	p_DSSMEMABConvStop		:= ADR(bConvStop);
	p_DSSMEMABDBA			:= ADR(bDBA);
	p_DSSMEMABDBAStat		:= ADR(bDBAStat);
	p_DSSMEMABTimer			:= ADR(bTimer);
	p_DSSMEMABVirtual		:= ADR(bVirtual);

	(* Always Change If Project Change *)

END_PROGRAM
```

### Pneu2SenInShutter.var - Change By Project
```iecst
(*2019-03-25*)
(**)
(*Action & State & Status*)
VAR
	p_Pneu2SenInShutterStat2 : UDINT;
	p_Pneu2SenInShutterStatus2 : UDINT;
	p_Pneu2SenInShutterStatTxt2 : UDINT;
END_VAR
(**)
(*Alarm*)
VAR
	p_Pneu2SenInShutterAlmData2 : UDINT;
END_VAR
(**)
(*Output*)
VAR
	p_Pneu2SenInShutterExtCtrl2 : UDINT;
	p_Pneu2SenInShutterRetCtrl2 : UDINT;
	p_Pneu2SenInShutterTwoCtrlOut2 : UDINT;
	p_Pneu2SenInShutterExtended2 : UDINT;
	p_Pneu2SenInShutterRetracted2 : UDINT;
END_VAR
```

### Program Logical/Pneu/Pneu2SenInShutter (IEC) - 1.00.0 - NtPneu v5.00.0

#### InputRef_Link.var
```iecst
(*2019-04-09*)
(**)
(*External*)
VAR
	p_bLinkOpsRun : REFERENCE TO BOOL;
END_VAR
(**)
VAR
	p_bLinkDISafetyRlySig : REFERENCE TO BOOL;
	p_bLinkDIPullerRetRS : REFERENCE TO BOOL;
	p_bLinkDIConvLftSen : REFERENCE TO BOOL;
END_VAR
```

#### Act_InitGlobal.st
```iecst
(** 2019-04-09 **)
ACTION Act_InitGlobal:

	(* Always Change If Project Change *)

	//Pass Data To Link
	p_bLinkOpsRun ACCESS p_OpsRun;

	p_bLinkDISafetyRlySig ACCESS p_DISafetyRlySig;
	p_bLinkDIPullerRetRS ACCESS p_DIPullerRetRS;
	p_bLinkDIConvLftSen ACCESS p_DIConvLftSen;

	//Pass Data To Internal Use
	p_udiRstErr ACCESS p_RstErrReset;
	p_bPrep ACCESS p_NtParamProjInletShutPrep;
	p_bManual ACCESS p_UIMnlMod;
	p_bSimu ACCESS p_UISimuMod;
	p_bTwoCtrlIn ACCESS p_NtParamInShutterTwoCtrlIn;
	p_sProgNm ACCESS p_NtParamInShutterProgNm;
	p_bExtSen ACCESS p_DIInShutterCloseRS;
	p_bRetSen ACCESS p_DIInShutterOpenRS;
	p_tExtTO ACCESS p_NtParamInShutterExtTO;
	p_tRetTO ACCESS p_NtParamInShutterRetTO;
	p_bNtSettingsLoadDone ACCESS p_StartupNtSettingsLoadDone;

	(* Always Change If Project Change *)

END_ACTION
```

#### Act_LinkAction.st
```iecst
(** 2019-04-09 **)
ACTION Act_LinkAction:

	IF p_bLinkOpsRun = TRUE THEN
		p_eAct ACCESS p_OpsTravLifLDInletPneuAct;
	ELSIF p_bManual = TRUE OR p_bSimu THEN
		p_eAct ACCESS p_UIInShutterAct;
	ELSE
		p_eAct ACCESS ADR(eAct);
	END_IF

END_ACTION
```

### Program Logical/Pneu/Pneu2SenOutShutter (IEC) - 1.00.0 - NtPneu v5.00.0

#### InputRef_Link.var
```iecst
(*2019-04-09*)
(**)
(*External*)
VAR
	p_bLinkOpsRun : REFERENCE TO BOOL;
END_VAR
(**)
VAR
	p_bLinkDISafetyRlySig : REFERENCE TO BOOL;
	p_bLinkInitOpsTravLifDone : REFERENCE TO BOOL;
	p_bLinkMcParamOutShutDis : REFERENCE TO BOOL;
	p_bLinkDIConvClrSen : REFERENCE TO BOOL;
END_VAR
```

#### Local.var
```iecst
(*2019-04-30*)
(**)
(*Local Action, State & Status*)
VAR
	eAct : ePneuAction := PneuActIdle;
	eStat : ePneuAction := PneuActIdle;
	eStatus : eFBStatus := Idle;
	udiStatus : UDINT := 0;
	sStatTxt : STRING[200] := '';
	a_sStatText : ARRAY[0..50] OF STRING[200] := ['Idling','Set All','Reset All','Set Extend','Set Retract','Extending','Retracting','Retracting From Extend Sensor To Middle Sensor','Retracting From Middle Sensor To Retract Sensor','Extending From Retract Sensor To Middle Sensor','Extending From Middle Sensor To Extend Sensor',40('')];
END_VAR
(**)
(*Local Alarm*)
VAR
	tyAlmData : tyAlmDat;
	a_tyAlmText : ARRAY[10000..10099] OF tyAlmTxt := [(sAlmText:='Safety Check Error While Extending',sRcyText:='Safety System Has Been Triggered. All Operations Are Disable. Remove the Obstacle That Triggered The Safety Interlock To Resume Operation.'),(sAlmText:='Extend Sensor On Checking Time Out While Extending',sRcyText:='Sensor Timeout Expired Before Operation Completed. Sensor Operation Is Abnormal. Solve The Error To Resume Operation. '),(sAlmText:='Retract Sensor Off Checking Time Out While Extending',sRcyText:='Sensor Timeout Expired Before Operation Completed. Sensor Operation Is Abnormal. Solve The Error To Resume Operation.'),(sAlmText:='Safety Check Error While Retracting',sRcyText:='Safety System Has Been Triggered. All Operations Are Disable. Remove the Obstacle That Triggered The Safety Interlock To Resume Operation.'),(sAlmText:='Retract Sensor On Checking Time Out While Retracting',sRcyText:='Sensor Timeout Expired Before Operation Completed. Sensor Operation Is Abnormal. Solve The Error To Resume Operation.'),(sAlmText:='Extend Sensor Off Checking Time Out While Retracting',sRcyText:='Sensor Timeout Expired Before Operation Completed. Sensor Operation Is Abnormal. Solve The Error To Resume Operation.'),94((0))];
END_VAR
(**)
(*Local Output*)
VAR
	bExtCtrl : BOOL;
	bRetCtrl : BOOL;
	bTwoCtrlOut : BOOL := FALSE;
	bExtended : BOOL := FALSE;
	bRetracted : BOOL := FALSE;
END_VAR
(**)
(*Local Input*)
VAR
	udiRstErr : UDINT := 0;
	bPrep : BOOL := TRUE;
	bEn : BOOL := TRUE;
	bDis : BOOL := FALSE;
	p_bSimu : REFERENCE TO BOOL;
	bManual : BOOL := FALSE;
	bTwoCtrlIn : BOOL := FALSE;
	bExtSafetySen : BOOL := TRUE;
	bRetSafetySen : BOOL := TRUE;
	bExtSen : BOOL := FALSE;
	bRetSen : BOOL := FALSE;
	sProgNm : STRING[15] := 'Pneu2Sen';
	tExtTO : TIME := T#20s;
	tRetTO : TIME := T#20s;
	bNtSettingsLoadDone : BOOL := TRUE;
END_VAR
(**)
(*Local*)
VAR
	bRstErr : BOOL;
	udiRstErrOld : UDINT;
	bInitDone : BOOL;
	bInitialDone : BOOL;
	fbPneuExtChk : fbPneuExtRetSenExtChk;
	fbPneuRetChk : fbPneuExtRetSenRetChk;
	eStatOld : ePneuAction := PneuActIdle;
	udiModuleNum : UDINT := 2551;
END_VAR
```

#### Act_InitGlobal.st
```iecst
(** 2019-04-09 **)
ACTION Act_InitGlobal:

	(* Always Change If Project Change *)

	//Pass Data To Link
	p_bLinkOpsRun ACCESS p_OpsRun;

	p_bLinkDISafetyRlySig ACCESS p_DISafetyRlySig;
	p_bLinkInitOpsTravLifDone ACCESS p_OpsTravLifLDInitDone;
	p_bLinkMcParamOutShutDis ACCESS p_McParamOutShutterDis;
	p_bLinkDIConvClrSen ACCESS p_DIConvClrSen;

	//Pass Data To Internal Use
	p_udiRstErr ACCESS p_RstErrReset;
	p_bPrep ACCESS p_NtParamProjOutletShutPrep;
//	p_bDis ACCESS p_McParamOutShutterDis;
	p_bSimu ACCESS p_UISimuMod;
	p_bManual ACCESS p_UIMnlMod;
	p_bTwoCtrlIn ACCESS p_NtParamOutShutterTwoCtrlIn;
	p_sProgNm ACCESS p_NtParamOutShutterProgNm;
	p_bExtSen ACCESS p_DIOutShutterCloseRS;
	p_bRetSen ACCESS p_DIOutShutterOpenRS;
	p_tExtTO ACCESS p_NtParamOutShutterExtTO;
	p_tRetTO ACCESS p_NtParamOutShutterRetTO;
	p_bNtSettingsLoadDone ACCESS p_StartupNtSettingsLoadDone;

	(* Always Change If Project Change *)

END_ACTION
```

#### Act_LinkAction.st
```iecst
(** 2019-04-09 **)
ACTION Act_LinkAction:

	IF p_bLinkOpsRun = TRUE THEN
		p_eAct ACCESS p_OpsTravLifLDOutletPneuAct;
	ELSIF p_bManual = TRUE OR p_bSimu THEN
		p_eAct ACCESS p_UIOutShutterAct;
	ELSE
		p_eAct ACCESS ADR(eAct);
	END_IF

END_ACTION
```

### Pneu2SenPuller.var - Change By Project
```iecst
(*2019-03-25*)
(**)
(*Action & State & Status*)
VAR
	p_Pneu2SenPullerStat : UDINT;
	p_Pneu2SenPullerStatus : UDINT;
	p_Pneu2SenPullerStatTxt : UDINT;
END_VAR
(**)
(*Alarm*)
VAR
	p_Pneu2SenPullerAlmData : UDINT;
END_VAR
(**)
(*Output*)
VAR
	p_Pneu2SenPullerExtCtrl : UDINT;
	p_Pneu2SenPullerRetCtrl : UDINT;
	p_Pneu2SenPullerTwoCtrlOut : UDINT;
	p_Pneu2SenPullerExtended : UDINT;
	p_Pneu2SenPullerRetracted : UDINT;
END_VAR
```

### Program Logical/Pneu/Pneu2SenPuller (IEC) - 1.00.0 - NtPneu v5.00.0

#### InputRef_Link.var
```iecst
(*2019-04-09*)
(**)
(*External*)
VAR
	p_bLinkOpsRun : REFERENCE TO BOOL;
END_VAR
(**)
VAR
	p_bLinkAlmErr : REFERENCE TO BOOL;
	p_bLinkDISafetyRlySig : REFERENCE TO BOOL;
END_VAR
```

#### Act_InitGlobal.st
```iecst
(** 2019-04-09 **)
ACTION Act_InitGlobal:

	(* Always Change If Project Change *)

	//Pass Data To Link
	p_bLinkOpsRun ACCESS p_OpsRun;

	p_bLinkAlmErr ACCESS p_AlarmErr;
	p_bLinkDISafetyRlySig ACCESS p_DISafetyRlySig;

	//Pass Data To Internal Use
	p_udiRstErr ACCESS p_RstErrReset;
	p_bDis ACCESS p_NtParamProjPullerRotCylPrep;
	p_bManual ACCESS p_UIMnlMod;
	p_bTwoCtrlIn ACCESS p_NtParamPullerTwoCtrlIn;
	p_sProgNm ACCESS p_NtParamPullerProgNm;
	p_bExtSen ACCESS p_DIPullerExtRS;
	p_bRetSen ACCESS p_DIPullerRetRS;
	p_tExtTO ACCESS p_NtParamPullerExtTO;
	p_tRetTO ACCESS p_NtParamPullerRetTO;
	p_bNtSettingsLoadDone ACCESS p_StartupNtSettingsLoadDone;

	(* Always Change If Project Change *)

END_ACTION
```

#### Act_Link.st
```iecst
(** 2019-03-29 **)
ACTION Act_Link:

	IF p_bLinkAlmErr OR NOT p_bLinkDISafetyRlySig THEN
		bExtCtrl	:= FALSE;
		bRetCtrl	:= FALSE;
		bExtended	:= FALSE;
		bRetracted	:= FALSE;
	END_IF

END_ACTION
```

#### Act_LinkAction.st
```iecst
(** 2019-04-09 **)
ACTION Act_LinkAction:

	IF p_bLinkOpsRun = TRUE THEN
		p_eAct ACCESS p_OpsTravLifLDPullerAct;
	ELSIF p_bManual = TRUE THEN
		p_eAct ACCESS p_UIPullerAct;
	ELSE
		p_eAct ACCESS ADR(eAct);
	END_IF

END_ACTION
```

#### Init.st
```iecst
(** 2019-03-25 **)
PROGRAM _INIT

	(* Always Change If Project Change *)

	//Pass Address To Global Address For External Use
	//Action, State & Status
	p_Pneu2SenPullerStat		:= ADR(eStat);
	p_Pneu2SenPullerStatus		:= ADR(eStatus);
	p_Pneu2SenPullerStatTxt		:= ADR(sStatTxt);

	//Alarm
	p_Pneu2SenPullerAlmData		:= ADR(tyAlmData);

	//Output
	p_Pneu2SenPullerExtCtrl		:= ADR(bExtCtrl);
	p_Pneu2SenPullerRetCtrl		:= ADR(bRetCtrl);
	p_Pneu2SenPullerTwoCtrlOut	:= ADR(bTwoCtrlOut);
	p_Pneu2SenPullerExtended	:= ADR(bExtended);
	p_Pneu2SenPullerRetracted	:= ADR(bRetracted);

	(* Always Change If Project Change *)

END_PROGRAM
```

### Program Logical/Pneu/SelClamp/Pneu2SenSelClamp1 (IEC) - 1.00.0 - NtPneu v5.00.0

#### Act_LinkAction.st
```iecst
(** 2019-04-09 **)
ACTION Act_LinkAction:

	IF p_bLinkOpsRun = TRUE THEN
		p_eAct ACCESS p_OpsMagConvLD1StepSelClampCtrl;
	ELSIF p_bManual = TRUE THEN
		p_eAct ACCESS p_UIMagConvSelClp1Act;
	ELSE
		p_eAct ACCESS ADR(eAct);
	END_IF

END_ACTION
```

### Program Logical/Pneu/SelClamp/Pneu2SenSelClamp2 (IEC) - 1.00.0 - NtPneu v5.00.0

#### Act_LinkAction.st
```iecst
(** 2019-04-09 **)
ACTION Act_LinkAction:

	IF p_bLinkOpsRun = TRUE THEN
		p_eAct ACCESS p_OpsMagConvLD2StepSelClampCtrl;
	ELSIF p_bManual = TRUE THEN
		p_eAct ACCESS p_UIMagConvSelClp2Act;
	ELSE
		p_eAct ACCESS ADR(eAct);
	END_IF

END_ACTION
```

### Program Logical/Pneu/SelClamp/Pneu2SenSelClamp3 (IEC) - 1.00.0 - NtPneu v5.00.0

#### Act_Alarm.st
```iecst
(** 2019-03-25 **)
ACTION Act_Alarm:

	//Error
	IF EDGEPOS(eStatus = Error) THEN

		tyAlmData.sProgNm		:= p_sProgNm;
		tyAlmData.udiCode		:= udiStatus;
		tyAlmData.eSeverity		:= AlmSeverityError;
		tyAlmData.udiRunTime	:= tyAlmData.udiRunTime + 1;
		tyAlmData.bAlm			:= TRUE;
		tyAlmData.udiModuleNum  := udiModuleNum;
		g_sPneu2SenProgNm		:= p_sProgNm;
		//Get Error Message
		IF tyAlmData.udiCode < 10000 OR tyAlmData.udiCode > 10099 THEN
			tyAlmData.sAlmMsg	:= 'Unknown';
			tyAlmData.sRcyMsg	:= 'Unknown';
		ELSE
			tyAlmData.sAlmMsg	:= a_tyAlmText[tyAlmData.udiCode].sAlmText;
			tyAlmData.sRcyMsg	:= a_tyAlmText[tyAlmData.udiCode].sRcyText;
		END_IF

		sStatTxt	:= tyAlmData.sAlmMsg;

	ELSIF bRstErr AND (tyAlmData.udiCode <> 0) THEN

		tyAlmData.udiCode	:= 0;
		tyAlmData.eSeverity	:= AlmSeverityNA;
		tyAlmData.sAlmMsg	:= '';
		tyAlmData.sRcyMsg	:= '';
		tyAlmData.bAlm			:= FALSE;
		sStatTxt	:= a_sStatText[eStat];

	END_IF

END_ACTION
```

#### Act_InitGlobal.st
```iecst
(** 2039-04-09 **)
ACTION Act_InitGlobal:

	(* Always Change If Project Change *)

	//Pass Data To Link
	p_bLinkOpsRun ACCESS p_OpsRun;

	p_bLinkDISafetyRlySig ACCESS p_DISafetyRlySig;

	//Pass Data To Internal Use
	p_udiRstErr ACCESS p_RstErrReset;
	p_bNtParamProjMagAutoVerifyPrep ACCESS p_NtParamProjMagAutoVerifyPrep;
	p_bManual ACCESS p_UIMnlMod;
	p_bTwoCtrlIn ACCESS p_NtParamSelClamp3TwoCtrlIn;
	p_sProgNm ACCESS p_NtParamSelClamp3ProgNm;
	p_bExtSen ACCESS p_DIMag3SelUnclampRS;
//	p_bRetSen ACCESS p_DIOutShutterOpenRS;
	p_tExtTO ACCESS p_NtParamSelClamp3ExtDlyTm;
	p_tRetTO ACCESS p_NtParamSelClamp3RetDlyTm;
	p_bNtSettingsLoadDone ACCESS p_StartupNtSettingsLoadDone;
	p_eProjMag ACCESS p_NtParamProjMag;
	(* Always Change If Project Change *)

END_ACTION
```

#### Act_LinkAction.st
```iecst
(** 2019-04-09 **)
ACTION Act_LinkAction:

	IF p_bLinkOpsRun = TRUE THEN
		p_eAct ACCESS p_OpsMagConvLD3StepSelClampCtrl;
	ELSIF p_bManual = TRUE THEN
		p_eAct ACCESS p_UIMagConvSelClp3Act;
	ELSE
		p_eAct ACCESS ADR(eAct);
	END_IF

END_ACTION
```

### Pneu2SenSelClamp4.var - Change By Project
```iecst
(*2039-03-25*)
(**)
(*Action & State & Status*)
VAR
	p_PneuNoSenSelClamp4Stat : UDINT;
	p_PneuNoSenSelClamp4Status : UDINT;
	p_PneuNoSenSelClamp4StatTxt : UDINT;
END_VAR
(**)
(*Alarm*)
VAR
	p_PneuNoSenSelClamp4AlmData : UDINT;
END_VAR
(**)
(*Output*)
VAR
	p_PneuNoSenSelClamp4ExtCtrl : UDINT;
	p_PneuNoSenSelClamp4RetCtrl : UDINT;
	p_PneuNoSenSelClamp4TwoCtrlOut : UDINT;
	p_PneuNoSenSelClamp4Extended : UDINT;
	p_PneuNoSenSelClamp4Retracted : UDINT;
END_VAR
```

### Program Logical/Pneu/SelClamp/Pneu2SenSelClamp4 (IEC) - 1.00.0 - NtPneu v5.00.0

#### InputRef.var
```iecst
(*2019-03-25*)
(**)
(*General*)
VAR
	p_eAct : REFERENCE TO ePneuAction;
	p_udiRstErr : REFERENCE TO UDINT;
	p_bPrep : REFERENCE TO BOOL;
	p_bEn : REFERENCE TO BOOL;
	p_bDis : REFERENCE TO BOOL;
END_VAR
(**)
(*Configuration*)
VAR
	p_bManual : REFERENCE TO BOOL;
	p_bTwoCtrlIn : REFERENCE TO BOOL;
	p_bExtSafetySen : REFERENCE TO BOOL;
	p_bRetSafetySen : REFERENCE TO BOOL;
	p_sProgNm : REFERENCE TO STRING[15];
	p_tExtTO : REFERENCE TO TIME;
	p_tRetTO : REFERENCE TO TIME;
	p_bNtSettingsLoadDone : REFERENCE TO BOOL;
	p_eProjMag : REFERENCE TO eLDMag;
	p_bNtParamProjMagAutoVerifyPrep : REFERENCE TO BOOL;
END_VAR
(**)
(*Input*)
VAR
	p_bExtSen : REFERENCE TO BOOL;
	p_bRetSen : REFERENCE TO BOOL;
END_VAR
```

#### Act_InitGlobal.st
```iecst
(** 2039-04-09 **)
ACTION Act_InitGlobal:

	(* Always Change If Project Change *)

	//Pass Data To Link
	p_bLinkOpsRun ACCESS p_OpsRun;

	p_bLinkDISafetyRlySig ACCESS p_DISafetyRlySig;

	//Pass Data To Internal Use
	p_udiRstErr ACCESS p_RstErrReset;
	p_bNtParamProjMagAutoVerifyPrep ACCESS p_NtParamProjMagAutoVerifyPrep;
	p_bManual ACCESS p_UIMnlMod;
	p_bTwoCtrlIn ACCESS p_NtParamSelClamp4TwoCtrlIn;
	p_sProgNm ACCESS p_NtParamSelClamp4ProgNm;
	p_bExtSen ACCESS p_DIMag4SelUnclampRS;
//	p_bRetSen ACCESS p_DIOutShutterOpenRS;
	p_tExtTO ACCESS p_NtParamSelClamp4ExtDlyTm;
	p_tRetTO ACCESS p_NtParamSelClamp4RetDlyTm;
	p_bNtSettingsLoadDone ACCESS p_StartupNtSettingsLoadDone;
	p_eProjMag ACCESS p_NtParamProjMag;
	(* Always Change If Project Change *)

END_ACTION
```

#### Act_Link.st
```iecst
(** 2019-03-29 **)
ACTION Act_Link:

	IF p_bLinkDISafetyRlySig = FALSE THEN
		bExtCtrl	:= FALSE;
		bRetCtrl	:= FALSE;
		bExtended	:= FALSE;
		bRetracted	:= FALSE;
	END_IF

	IF (p_bPrep = TRUE) AND (p_bEn = TRUE) AND (p_bDis = FALSE) THEN
		p_bRetSen := NOT(p_bExtSen);
	ELSE
		p_bRetSen := FALSE;
	END_IF

END_ACTION
```

#### Act_LinkAction.st
```iecst
(** 2019-04-09 **)
ACTION Act_LinkAction:

	IF p_bLinkOpsRun = TRUE THEN
		p_eAct ACCESS p_OpsMagConvLD4StepSelClampCtrl;
	ELSIF p_bManual = TRUE THEN
		p_eAct ACCESS p_UIMagConvSelClp4Act;
	ELSE
		p_eAct ACCESS ADR(eAct);
	END_IF

END_ACTION
```

#### Act_LinkEn.st
```iecst
(** 2019-01-11 **)
ACTION Act_LinkEn:

	//Link bPrep, bEn & bDis
	IF p_eProjMag = LDMagDual  THEN
		p_bPrep := FALSE;
	ELSIF p_eProjMag = LDMagTriple AND p_bNtParamProjMagAutoVerifyPrep THEN
		p_bPrep := TRUE;
	ELSE
		p_bPrep := FALSE;
	END_IF

END_ACTION
```

#### Init.st
```iecst
(** 2039-03-25 **)
PROGRAM _INIT

	(* Always Change If Project Change *)

	//Pass Address To Global Address For External Use
	//Action, State & Status
	p_PneuNoSenSelClamp4Stat		:= ADR(eStat);
	p_PneuNoSenSelClamp4Status		:= ADR(eStatus);
	p_PneuNoSenSelClamp4StatTxt		:= ADR(sStatTxt);

	//Alarm
	p_PneuNoSenSelClamp4AlmData		:= ADR(tyAlmData);

	//Output
	p_PneuNoSenSelClamp4ExtCtrl		:= ADR(bExtCtrl);
	p_PneuNoSenSelClamp4RetCtrl		:= ADR(bRetCtrl);
	p_PneuNoSenSelClamp4TwoCtrlOut	:= ADR(bTwoCtrlOut);
	p_PneuNoSenSelClamp4Extended	:= ADR(bExtended);
	p_PneuNoSenSelClamp4Retracted	:= ADR(bRetracted);

	(* Always Change If Project Change *)

END_PROGRAM
```

### Program Logical/Pneu/MagSafetyBar/Pneu2SenMag1SafetyBar (IEC) - 1.00.0 - NtPneu v5.00.0

#### InputRef_Link.var
```iecst
(*2019-04-09*)
(**)
(*External*)
VAR
	p_bLinkOpsRun : REFERENCE TO BOOL;
END_VAR
(**)
VAR
	p_bLinkDISafetyRlySig : REFERENCE TO BOOL;
	p_bLinkNtPrmProjMagSafetyBarPrep : REFERENCE TO BOOL;
	p_bLinkMagSafetyBarDisabledFront : REFERENCE TO BOOL;
	p_bLinkMagSafetyBarDisabledRear : REFERENCE TO BOOL;
END_VAR
```

#### Act_Alarm.st
```iecst
(** 2019-03-25 **)
ACTION Act_Alarm:

	//Error
	IF EDGEPOS(eStatus = Error) THEN

		tyAlmData.sProgNm		:= p_sProgNm;
		tyAlmData.udiCode		:= udiStatus;
		tyAlmData.eSeverity		:= AlmSeverityError;
		tyAlmData.udiRunTime	:= tyAlmData.udiRunTime + 1;
		tyAlmData.bAlm			:= TRUE;
		tyAlmData.udiModuleNum  := udiModuleNum;
		g_sPneu2SenProgNm		:= p_sProgNm;
		//Get Error Message
		IF tyAlmData.udiCode < 10000 OR tyAlmData.udiCode > 10099 THEN
			tyAlmData.sAlmMsg	:= 'Unknown';
			tyAlmData.sRcyMsg	:= 'Unknown';
		ELSE
			tyAlmData.sAlmMsg	:= a_tyAlmText[tyAlmData.udiCode].sAlmText;
			tyAlmData.sRcyMsg	:= a_tyAlmText[tyAlmData.udiCode].sRcyText;
		END_IF

		sStatTxt	:= tyAlmData.sAlmMsg;

	ELSIF bRstErr AND (tyAlmData.udiCode <> 0) THEN

		tyAlmData.udiCode	:= 0;
		tyAlmData.eSeverity	:= AlmSeverityNA;
		tyAlmData.sAlmMsg	:= '';
		tyAlmData.sRcyMsg	:= '';
		tyAlmData.bAlm			:= FALSE;
		sStatTxt	:= a_sStatText[eStat];

	END_IF

END_ACTION
```

#### Act_InitGlobal.st
```iecst
(** 2019-04-09 **)
ACTION Act_InitGlobal:

	(* Always Change If Project Change *)

	//Pass Data To Link
	p_bLinkOpsRun ACCESS p_OpsRun;

	p_bLinkNtPrmProjMagSafetyBarPrep ACCESS p_NtParamProjMagSafetyBarPrep;
	p_bLinkDISafetyRlySig ACCESS p_DISafetyRlySig;
	p_bLinkMagSafetyBarDisabledFront ACCESS p_MagRcpCurrRcpSBarDisabled;
	p_bLinkMagSafetyBarDisabledRear ACCESS p_MagRcpCurrRcpSBarDisabled1;

	p_eLinkMag ACCESS p_NtParamProjMag;
	p_usiLinkMod ACCESS p_ProdRcpCurrRcp1McMod;
	//Pass Data To Internal Use
	p_udiRstErr ACCESS p_RstErrReset;
	p_bPrep ACCESS p_NtParamProjMagSafetyBarPrep;
	p_bManual ACCESS p_UIMnlMod;
	p_bTwoCtrlIn ACCESS p_NtParamMag1SafetyBarTwoCtrlIn;
	p_sProgNm ACCESS p_NtParamMag1SafetyBarProgNm;
	p_bExtSen ACCESS p_DIMag1SafetyBarExtRS;
	p_bRetSen ACCESS p_DIMag1SafetyBarRetRS;
	p_tExtTO ACCESS p_NtParamMag1SafetyBarExtTO;
	p_tRetTO ACCESS p_NtParamMag1SafetyBarRetTO;
	p_bNtSettingsLoadDone ACCESS p_StartupNtSettingsLoadDone;

	p_eLinkMag ACCESS p_NtParamProjMag;
	p_usiLinkMod ACCESS p_ProdRcpCurrRcp1McMod;
	(* Always Change If Project Change *)

END_ACTION
```

#### Act_LinkAction.st
```iecst
(** 2019-04-09 **)
ACTION Act_LinkAction:

	IF p_bLinkOpsRun = TRUE THEN
		p_eAct ACCESS p_OpsMagConvLD1SafetyBarAct;
	ELSIF p_bManual = TRUE THEN
		p_eAct ACCESS p_UIMag1SafetyBarAct;
	ELSE
		p_eAct ACCESS ADR(eAct);
	END_IF

END_ACTION
```

#### Act_LinkEn.st
```iecst
(** 2019-01-11 **)
ACTION Act_LinkEn:

	//Link bPrep, bEn & bDis
	p_bPrep	:= p_bLinkNtPrmProjMagSafetyBarPrep;

	IF p_bLinkOpsRun AND p_bPrep THEN
		IF p_eLinkMag = LDMagQuadruple THEN
			CASE p_usiLinkMod OF
				0: //LDModLoadLnA:
					p_bDis := p_bLinkMagSafetyBarDisabledFront;
				1: //LDModLoadLnB:
					p_bDis := p_bLinkMagSafetyBarDisabledRear;

				2: //LDModLoadLnAB:
					p_bDis := p_bLinkMagSafetyBarDisabledFront;

			END_CASE
		ELSE
			p_bDis := p_bLinkMagSafetyBarDisabledFront;

		END_IF
	END_IF

END_ACTION
```

### Program Logical/Pneu/MagSafetyBar/Pneu2SenMag2SafetyBar (IEC) - 1.00.0 - NtPneu v5.00.0

#### InputRef.var
```iecst
(*2019-03-25*)
(**)
(*General*)
VAR
	p_eAct : REFERENCE TO ePneuAction;
	p_udiRstErr : REFERENCE TO UDINT;
	p_bPrep : REFERENCE TO BOOL;
	p_bEn : REFERENCE TO BOOL;
	p_bDis : REFERENCE TO BOOL;
END_VAR
(**)
(*Configuration*)
VAR
	p_bManual : REFERENCE TO BOOL;
	p_bTwoCtrlIn : REFERENCE TO BOOL;
	p_bExtSafetySen : REFERENCE TO BOOL;
	p_bRetSafetySen : REFERENCE TO BOOL;
	p_sProgNm : REFERENCE TO STRING[15];
	p_tExtTO : REFERENCE TO TIME;
	p_tRetTO : REFERENCE TO TIME;
	p_bNtSettingsLoadDone : REFERENCE TO BOOL;
	p_eLinkMag : REFERENCE TO eLDMag;
	p_usiLinkMod : REFERENCE TO USINT;
END_VAR
(**)
(*Input*)
VAR
	p_bExtSen : REFERENCE TO BOOL;
	p_bRetSen : REFERENCE TO BOOL;
END_VAR
```

#### Act_InitGlobal.st
```iecst
(** 2019-04-09 **)
ACTION Act_InitGlobal:

	(* Always Change If Project Change *)

	//Pass Data To Link
	p_bLinkOpsRun ACCESS p_OpsRun;

	p_bLinkNtPrmProjMagSafetyBarPrep ACCESS p_NtParamProjMagSafetyBarPrep;
	p_bLinkDISafetyRlySig ACCESS p_DISafetyRlySig;
	p_bLinkMagSafetyBarDisabledFront ACCESS p_MagRcpCurrRcpSBarDisabled;
	p_bLinkMagSafetyBarDisabledRear ACCESS p_MagRcpCurrRcpSBarDisabled1;

	p_eLinkMag ACCESS p_NtParamProjMag;
	p_usiLinkMod ACCESS p_ProdRcpCurrRcp1McMod;
	//Pass Data To Internal Use
	p_udiRstErr ACCESS p_RstErrReset;
	p_bPrep ACCESS p_NtParamProjMagSafetyBarPrep;
	p_bManual ACCESS p_UIMnlMod;
	p_bTwoCtrlIn ACCESS p_NtParamMag2SafetyBarTwoCtrlIn;
	p_sProgNm ACCESS p_NtParamMag2SafetyBarProgNm;
	p_bExtSen ACCESS p_DIMag2SafetyBarExtRS;
	p_bRetSen ACCESS p_DIMag2SafetyBarRetRS;
	p_tExtTO ACCESS p_NtParamMag2SafetyBarExtTO;
	p_tRetTO ACCESS p_NtParamMag2SafetyBarRetTO;
	p_bNtSettingsLoadDone ACCESS p_StartupNtSettingsLoadDone;

	(* Always Change If Project Change *)

END_ACTION
```

#### Act_LinkAction.st
```iecst
(** 2019-04-09 **)
ACTION Act_LinkAction:

	IF p_bLinkOpsRun = TRUE THEN
		p_eAct ACCESS p_OpsMagConvLD2SafetyBarAct;
	ELSIF p_bManual = TRUE THEN
		p_eAct ACCESS p_UIMag2SafetyBarAct;
	ELSE
		p_eAct ACCESS ADR(eAct);
	END_IF

END_ACTION
```

#### Act_LinkEn.st
```iecst
(** 2019-01-11 **)
ACTION Act_LinkEn:

	//Link bPrep, bEn & bDis
	p_bPrep	:= p_bLinkNtPrmProjMagSafetyBarPrep;

	IF p_bLinkOpsRun AND p_bPrep THEN
		IF p_eLinkMag = LDMagQuadruple THEN
			CASE p_usiLinkMod OF
				0: //LDModLoadLnA:
					p_bDis := p_bLinkMagSafetyBarDisabledFront;
				1: //LDModLoadLnB:
					p_bDis := p_bLinkMagSafetyBarDisabledRear;

				2: //LDModLoadLnAB:
					p_bDis := p_bLinkMagSafetyBarDisabledFront;

			END_CASE
		ELSE
			p_bDis := p_bLinkMagSafetyBarDisabledFront;

		END_IF
	END_IF

END_ACTION
```

### Program Logical/Pneu/MagSafetyBar/Pneu2SenMag3SafetyBar (IEC) - 1.00.0 - NtPneu v5.00.0

#### InputRef.var
```iecst
(*2019-03-25*)
(**)
(*General*)
VAR
	p_eAct : REFERENCE TO ePneuAction;
	p_udiRstErr : REFERENCE TO UDINT;
	p_bPrep : REFERENCE TO BOOL;
	p_bEn : REFERENCE TO BOOL;
	p_bDis : REFERENCE TO BOOL;
END_VAR
(**)
(*Configuration*)
VAR
	p_bManual : REFERENCE TO BOOL;
	p_bTwoCtrlIn : REFERENCE TO BOOL;
	p_bExtSafetySen : REFERENCE TO BOOL;
	p_bRetSafetySen : REFERENCE TO BOOL;
	p_sProgNm : REFERENCE TO STRING[15];
	p_tExtTO : REFERENCE TO TIME;
	p_tRetTO : REFERENCE TO TIME;
	p_bNtSettingsLoadDone : REFERENCE TO BOOL;
	p_eProjMag : REFERENCE TO eLDMag;
	p_eLinkMag : REFERENCE TO eLDMag;
	p_usiLinkMod : REFERENCE TO USINT;
END_VAR
(**)
(*Input*)
VAR
	p_bExtSen : REFERENCE TO BOOL;
	p_bRetSen : REFERENCE TO BOOL;
END_VAR
```

#### Act_InitGlobal.st
```iecst
(** 2019-04-09 **)
ACTION Act_InitGlobal:

	(* Always Change If Project Change *)

	//Pass Data To Link
	p_bLinkOpsRun ACCESS p_OpsRun;

	p_bLinkNtPrmProjMagSafetyBarPrep ACCESS p_NtParamProjMagSafetyBarPrep;
	p_bLinkNtPrmProjMag ACCESS p_NtParamProjMag;

	p_bLinkDISafetyRlySig ACCESS p_DISafetyRlySig;
	p_bLinkMagSafetyBarDisabledFront ACCESS p_MagRcpCurrRcpSBarDisabled;
	p_bLinkMagSafetyBarDisabledRear ACCESS p_MagRcpCurrRcpSBarDisabled1;

	p_eLinkMag ACCESS p_NtParamProjMag;
	p_usiLinkMod ACCESS p_ProdRcpCurrRcp1McMod;
	//Pass Data To Internal Use
	p_udiRstErr ACCESS p_RstErrReset;
	p_bManual ACCESS p_UIMnlMod;
	p_bTwoCtrlIn ACCESS p_NtParamMag3SafetyBarTwoCtrlIn;
	p_sProgNm ACCESS p_NtParamMag3SafetyBarProgNm;
	p_bExtSen ACCESS p_DIMag3SafetyBarExtRS;
	p_bRetSen ACCESS p_DIMag3SafetyBarRetRS;
	p_tExtTO ACCESS p_NtParamMag3SafetyBarExtTO;
	p_tRetTO ACCESS p_NtParamMag3SafetyBarRetTO;
	p_bNtSettingsLoadDone ACCESS p_StartupNtSettingsLoadDone;
	p_eProjMag ACCESS p_NtParamProjMag;
	(* Always Change If Project Change *)

END_ACTION
```

#### Act_LinkAction.st
```iecst
(** 2019-04-09 **)
ACTION Act_LinkAction:

	IF p_bLinkOpsRun = TRUE THEN
		p_eAct ACCESS p_OpsMagConvLD3SafetyBarAct;
	ELSIF p_bManual = TRUE THEN
		p_eAct ACCESS p_UIMag3SafetyBarAct;
	ELSE
		p_eAct ACCESS ADR(eAct);
	END_IF

END_ACTION
```

#### Act_LinkEn.st
```iecst
(** 2019-01-11 **)
ACTION Act_LinkEn:

	//Link bPrep, bEn & bDis
	p_bPrep	:= p_bLinkNtPrmProjMagSafetyBarPrep AND p_bLinkNtPrmProjMag = LDMagTriple;

	IF p_bLinkOpsRun AND p_bPrep THEN
		IF p_eLinkMag = LDMagQuadruple THEN
			CASE p_usiLinkMod OF
				0: //LDModLoadLnA:
					p_bDis := p_bLinkMagSafetyBarDisabledFront;
				1: //LDModLoadLnB:
					p_bDis := p_bLinkMagSafetyBarDisabledRear;

				2: //LDModLoadLnAB:
					p_bDis := p_bLinkMagSafetyBarDisabledRear;

			END_CASE
		ELSE
			p_bDis := p_bLinkMagSafetyBarDisabledFront;

		END_IF
	END_IF

END_ACTION
```

### Pneu2SenMag4SafetyBar.var - Change By Project
```iecst
(*2019-03-25*)
(**)
(*Action & State & Status*)
VAR
	p_Pneu2SMag4SafetyBarStat : UDINT;
	p_Pneu2SMag4SafetyBarStatus : UDINT;
	p_Pneu2SMag4SafetyBarStatTxt : UDINT;
END_VAR
(**)
(*Alarm*)
VAR
	p_Pneu2SMag4SafetyBarAlmData : UDINT;
END_VAR
(**)
(*Output*)
VAR
	p_Pneu2SMag4SafetyBarExtCtrl : UDINT;
	p_Pneu2SMag4SafetyBarRetCtrl : UDINT;
	p_Pneu2SMag4SafetyBarTwoCtrlOut : UDINT;
	p_Pneu2SMag4SafetyBarExtended : UDINT;
	p_Pneu2SMag4SafetyBarRetracted : UDINT;
END_VAR
```

### Program Logical/Pneu/MagSafetyBar/Pneu2SenMag4SafetyBar (IEC) - 1.00.0 - NtPneu v5.00.0

#### InputRef_Link.var
```iecst
(*2019-04-09*)
(**)
(*External*)
VAR
	p_bLinkOpsRun : REFERENCE TO BOOL;
END_VAR
(**)
VAR
	p_bLinkNtPrmProjMagSafetyBarPrep : REFERENCE TO BOOL;
	p_bLinkNtPrmProjMag : REFERENCE TO eLDMag;
END_VAR
(**)
VAR
	p_bLinkDISafetyRlySig : REFERENCE TO BOOL;
	p_bLinkMagSafetyBarDisabledFront : REFERENCE TO BOOL;
	p_bLinkMagSafetyBarDisabledRear : REFERENCE TO BOOL;
END_VAR
```

#### Act_Alarm.st
```iecst
(** 2019-03-25 **)
ACTION Act_Alarm:

	//Error
	IF EDGEPOS(eStatus = Error) THEN

		tyAlmData.sProgNm		:= p_sProgNm;
		tyAlmData.udiCode		:= udiStatus;
		tyAlmData.eSeverity		:= AlmSeverityError;
		tyAlmData.udiRunTime	:= tyAlmData.udiRunTime + 1;
		tyAlmData.bAlm			:= TRUE;
		tyAlmData.udiModuleNum  := udiModuleNum;
		g_sPneu2SenProgNm		:= p_sProgNm;
		//Get Error Message
		IF tyAlmData.udiCode < 10000 OR tyAlmData.udiCode > 10099 THEN
			tyAlmData.sAlmMsg	:= 'Unknown';
			tyAlmData.sRcyMsg	:= 'Unknown';
		ELSE
			tyAlmData.sAlmMsg	:= a_tyAlmText[tyAlmData.udiCode].sAlmText;
			tyAlmData.sRcyMsg	:= a_tyAlmText[tyAlmData.udiCode].sRcyText;
		END_IF

		sStatTxt	:= tyAlmData.sAlmMsg;

	ELSIF bRstErr AND (tyAlmData.udiCode <> 0) THEN

		tyAlmData.udiCode	:= 0;
		tyAlmData.eSeverity	:= AlmSeverityNA;
		tyAlmData.sAlmMsg	:= '';
		tyAlmData.sRcyMsg	:= '';
		tyAlmData.bAlm			:= FALSE;
		sStatTxt	:= a_sStatText[eStat];

	END_IF

END_ACTION
```

#### Act_InitGlobal.st
```iecst
(** 2019-04-09 **)
ACTION Act_InitGlobal:

	(* Always Change If Project Change *)

	//Pass Data To Link
	p_bLinkOpsRun ACCESS p_OpsRun;

	p_bLinkNtPrmProjMagSafetyBarPrep ACCESS p_NtParamProjMagSafetyBarPrep;
	p_bLinkNtPrmProjMag ACCESS p_NtParamProjMag;

	p_bLinkDISafetyRlySig ACCESS p_DISafetyRlySig;
	p_bLinkMagSafetyBarDisabledFront ACCESS p_MagRcpCurrRcpSBarDisabled;
	p_bLinkMagSafetyBarDisabledRear ACCESS p_MagRcpCurrRcpSBarDisabled1;

	p_eLinkMag ACCESS p_NtParamProjMag;
	p_usiLinkMod ACCESS p_ProdRcpCurrRcp1McMod;

	//Pass Data To Internal Use
	p_udiRstErr ACCESS p_RstErrReset;
	p_bManual ACCESS p_UIMnlMod;
	p_bTwoCtrlIn ACCESS p_NtParamMag3SafetyBarTwoCtrlIn;
	p_sProgNm ACCESS p_NtParamMag3SafetyBarProgNm;
	p_bExtSen ACCESS p_DIMag4SafetyBarExtRS;
	p_bRetSen ACCESS p_DIMag4SafetyBarRetRS;
	p_tExtTO ACCESS p_NtParamMag4SafetyBarExtTO;
	p_tRetTO ACCESS p_NtParamMag4SafetyBarRetTO;
	p_bNtSettingsLoadDone ACCESS p_StartupNtSettingsLoadDone;

	(* Always Change If Project Change *)

END_ACTION
```

#### Act_LinkAction.st
```iecst
(** 2019-04-09 **)
ACTION Act_LinkAction:

	IF p_bLinkOpsRun = TRUE THEN
		p_eAct ACCESS p_OpsMagConvLD4SafetyBarAct;
	ELSIF p_bManual = TRUE THEN
//		p_eAct ACCESS p_UIMag4SafetyBarAct;
	ELSE
		p_eAct ACCESS ADR(eAct);
	END_IF

END_ACTION
```

#### Act_LinkEn.st
```iecst
(** 2019-01-11 **)
ACTION Act_LinkEn:

	//Link bPrep, bEn & bDis
	p_bPrep	:= p_bLinkNtPrmProjMagSafetyBarPrep AND p_bLinkNtPrmProjMag = LDMagQuadruple;

	IF p_bLinkOpsRun AND p_bPrep THEN
		IF p_eLinkMag = LDMagQuadruple THEN
			CASE p_usiLinkMod OF
				0: //LDModLoadLnA:
					p_bDis := p_bLinkMagSafetyBarDisabledFront;
				1: //LDModLoadLnB:
					p_bDis := p_bLinkMagSafetyBarDisabledRear;

				2: //LDModLoadLnAB:
					p_bDis := p_bLinkMagSafetyBarDisabledRear;

			END_CASE
		ELSE
			p_bDis := p_bLinkMagSafetyBarDisabledFront;

		END_IF
	END_IF

END_ACTION
```

#### Init.st
```iecst
(** 2019-03-25 **)
PROGRAM _INIT

	(* Always Change If Project Change *)

	//Pass Address To Global Address For External Use
	//Action, State & Status
	p_Pneu2SMag4SafetyBarStat		:= ADR(eStat);
	p_Pneu2SMag4SafetyBarStatus		:= ADR(eStatus);
	p_Pneu2SMag4SafetyBarStatTxt	:= ADR(sStatTxt);

	//Alarm
	p_Pneu2SMag4SafetyBarAlmData	:= ADR(tyAlmData);

	//Output
	p_Pneu2SMag4SafetyBarExtCtrl	:= ADR(bExtCtrl);
	p_Pneu2SMag4SafetyBarRetCtrl	:= ADR(bRetCtrl);
	p_Pneu2SMag4SafetyBarTwoCtrlOut	:= ADR(bTwoCtrlOut);
	p_Pneu2SMag4SafetyBarExtended	:= ADR(bExtended);
	p_Pneu2SMag4SafetyBarRetracted	:= ADR(bRetracted);

	(* Always Change If Project Change *)

END_PROGRAM
```

### PneuExtSenTrolley.var - Change By Project
```iecst
(*2019-03-25*)
(**)
(*Action & State & Status*)
VAR
	p_PneuExtSenTrllyStat : UDINT;
	p_PneuExtSenTrllyStatus : UDINT;
	p_PneuExtSenTrllyStatTxt : UDINT;
END_VAR
(**)
(*Alarm*)
VAR
	p_PneuExtSenTrllyAlmData : UDINT;
END_VAR
(**)
(*Output*)
VAR
	p_PneuExtSenTrllyExtCtrl : UDINT;
	p_PneuExtSenTrllyRetCtrl : UDINT;
	p_PneuExtSenTrllyTwoCtrlOut : UDINT;
	p_PneuExtSenTrllyExtended : UDINT;
	p_PneuExtSenTrllyRetracted : UDINT;
END_VAR
```

### Program Logical/Pneu/Trolley/PneuExtSenTrolley (IEC, version 1.00.0) - 1.00.0 - NtPneu v5.00.0

#### Init.st - Change By Project
```iecst
(** 2019-03-25 **)
PROGRAM _INIT

	(* Always Change If Project Change *)

	//Pass Address To Global Address For External Use
	//Action, State & Status
	p_PneuExtSenTrllyStat		:= ADR(eStat);
	p_PneuExtSenTrllyStatus		:= ADR(eStatus);
	p_PneuExtSenTrllyStatTxt		:= ADR(sStatTxt);

	//Alarm
	p_PneuExtSenTrllyAlmData		:= ADR(tyAlmData);

	//Output
	p_PneuExtSenTrllyExtCtrl		:= ADR(bExtCtrl);
	p_PneuExtSenTrllyRetCtrl		:= ADR(bRetCtrl);
	p_PneuExtSenTrllyTwoCtrlOut		:= ADR(bTwoCtrlOut);
	p_PneuExtSenTrllyExtended		:= ADR(bExtended);
	p_PneuExtSenTrllyRetracted		:= ADR(bRetracted);

	(* Always Change If Project Change *)

END_PROGRAM
```

#### Act_InitGlobal.st - Change By Project
```iecst
(** 2019-04-09 **)
ACTION Act_InitGlobal:

	(* Always Change If Project Change *)

	//Pass Data To Link
	p_bLinkOpsRun ACCESS p_OpsRun;
	p_bLinkDISafetyRlySig ACCESS p_DISafetyRlySig;

	//Pass Data To Internal Use
	p_bPrep ACCESS p_NtParamTrolleyLckPrep;
	p_bExtSen ACCESS p_DITrolleyExtRS1;
	p_tRetTO ACCESS p_NtParamTrolleyLckRetTO;
	p_tExtTO ACCESS p_NtParamTrolleyLckExtTO;
	p_bTwoCtrlIn ACCESS p_NtParamTrolleyLckTwoCtrlIn;

	p_udiRstErr ACCESS p_RstErrReset;
	p_bManual ACCESS p_UIMnlMod;
	p_bNtSettingsLoadDone ACCESS p_StartupNtSettingsLoadDone;

	(* Always Change If Project Change *)

END_ACTION
```

#### InputRef_Link.var - Change By Project
```iecst
(*2019-04-09*)
(**)
VAR
	p_bLinkOpsRun : REFERENCE TO BOOL;
	p_bLinkDISafetyRlySig : REFERENCE TO BOOL;
END_VAR
```

#### Act_LinkAction.st - Change By Project
```iecst
(** 2019-04-09 **)
ACTION Act_LinkAction:

	IF p_bLinkOpsRun = TRUE THEN
		p_eAct ACCESS p_OpsMagConvLD1TrolleyLck;
	ELSIF p_bManual = TRUE THEN
		p_eAct ACCESS p_UITrolleyLckAct1;
	ELSE
		p_eAct ACCESS ADR(eAct);
	END_IF

END_ACTION
```

#### Act_InitLocal.st - Do Not Change!!!
```iecst
(** 2019-03-25 **)
ACTION Act_InitLocal:

	//Input Reference Link To Local Variable
	p_eAct ACCESS ADR(eAct);
	p_udiRstErr ACCESS ADR(udiRstErr);
	p_bPrep ACCESS ADR(bPrep);
	p_bEn ACCESS ADR(bEn);
	p_bDis ACCESS ADR(bDis);
	p_bManual ACCESS ADR(bManual);
	p_bTwoCtrlIn ACCESS ADR(bTwoCtrlIn);
	p_bExtSafetySen ACCESS ADR(bExtSafetySen);
	p_bRetSafetySen ACCESS ADR(bRetSafetySen);
	p_sProgNm ACCESS ADR(sProgNm);
	p_tExtTO ACCESS ADR(tExtTO);
	p_tRetTO ACCESS ADR(tRetTO);
	p_bNtSettingsLoadDone ACCESS ADR(bNtSettingsLoadDone);
	p_bExtSen ACCESS ADR(bExtSen);

END_ACTION
```
